LIN {X 0.112,Y -477.429,Z 574.534,A 0.000,B 0.000,C 90.000,E1 96.144} C_DIS
LIN {X 0.154,Y -458.820,Z 574.520,A 0.000,B 0.000,C 90.000,E1 93.612} C_DIS
LIN {X 0.164,Y -448.919,Z 574.512,A 0.000,B 0.000,C 90.000,E1 92.064} C_DIS
LIN {X -0.078,Y -437.148,Z 574.500,A 0.000,B 0.000,C 90.000,E1 90.000} C_DIS
LIN {X -0.153,Y -429.554,Z 574.493,A 0.000,B 0.000,C 90.000,E1 88.682} C_DIS
LIN {X -0.207,Y -419.996,Z 574.484,A 0.000,B 0.000,C 90.000,E1 87.078} C_DIS
LIN {X -0.150,Y -405.811,Z 574.470,A 0.000,B 0.000,C 90.000,E1 84.609} C_DIS
LIN {X 0.053,Y -392.137,Z 574.456,A 0.000,B 0.000,C 90.000,E1 82.064} C_DIS
LIN {X -0.071,Y -380.234,Z 574.443,A 0.000,B 0.000,C 90.000,E1 79.803} C_DIS
LIN {X 0.033,Y -369.905,Z 574.432,A 0.000,B 0.000,C 90.000,E1 77.757} C_DIS
LIN {X -0.039,Y -355.862,Z 574.416,A 0.000,B 0.000,C 90.000,E1 74.810} C_DIS
LIN {X 0.162,Y -345.723,Z 574.402,A 0.000,B 0.000,C 90.000,E1 72.362} C_DIS
LIN {X -0.128,Y -334.343,Z 574.385,A 0.000,B 0.000,C 90.000,E1 69.337} C_DIS
LIN {X 0.102,Y -322.277,Z 574.364,A 0.000,B 0.000,C 90.000,E1 65.537} C_DIS
LIN {X 0.039,Y -314.723,Z 574.350,A 0.000,B 0.000,C 90.000,E1 62.999} C_DIS
LIN {X 0.116,Y -309.189,Z 574.339,A 0.000,B 0.000,C 90.000,E1 61.051} C_DIS
LIN {X 0.043,Y -301.821,Z 574.325,A 0.000,B 0.000,C 90.000,E1 58.456} C_DIS
LIN {X -0.131,Y -293.043,Z 574.306,A 0.000,B 0.000,C 90.000,E1 55.182} C_DIS
LIN {X -0.027,Y -286.344,Z 574.292,A 0.000,B 0.000,C 90.000,E1 52.477} C_DIS
LIN {X -0.003,Y -281.279,Z 574.280,A 0.000,B 0.000,C 90.000,E1 50.436} C_DIS
LIN {X 0.057,Y -277.727,Z 574.273,A 0.000,B 0.000,C 90.000,E1 49.057} C_DIS
LIN {X -0.110,Y -273.909,Z 574.265,A 0.000,B 0.000,C 90.000,E1 47.715} C_DIS
LIN {X 0.043,Y -269.773,Z 574.257,A 0.000,B 0.000,C 90.000,E1 46.296} C_DIS
LIN {X 0.008,Y -264.223,Z 574.248,A 0.000,B 0.000,C 90.000,E1 44.555} C_DIS
LIN {X -0.039,Y -256.042,Z 574.234,A 0.000,B 0.000,C 90.000,E1 42.081} C_DIS
LIN {X -0.053,Y -247.040,Z 574.218,A 0.000,B 0.000,C 90.000,E1 39.197} C_DIS
LIN {X -0.005,Y -238.686,Z 574.201,A 0.000,B 0.000,C 90.000,E1 36.251} C_DIS
LIN {X -0.102,Y -231.066,Z 574.185,A 0.000,B 0.000,C 90.000,E1 33.293} C_DIS
LIN {X -0.069,Y -224.084,Z 574.168,A 0.000,B 0.000,C 90.000,E1 30.256} C_DIS
LIN {X -0.051,Y -217.874,Z 574.151,A 0.000,B 0.000,C 90.000,E1 27.180} C_DIS
LIN {X 0.042,Y -211.020,Z 574.129,A 0.000,B 0.000,C 90.000,E1 23.259} C_DIS
LIN {X -0.047,Y -207.521,Z 574.116,A 0.000,B 0.000,C 90.000,E1 20.918} C_DIS
LIN {X 0.044,Y -203.153,Z 574.094,A 0.000,B 0.000,C 90.000,E1 16.913} C_DIS
LIN {X -0.057,Y -199.050,Z 574.067,A 0.000,B 0.000,C 90.000,E1 12.119} C_DIS
LIN {X -0.009,Y -196.173,Z 574.036,A 0.000,B 0.000,C 90.000,E1 6.429} C_DIS
LIN {X 0.096,Y -197.227,Z 573.966,A 0.000,B 0.000,C 90.000,E1 353.799} C_DIS
LIN {X 0.117,Y -200.242,Z 573.939,A 0.000,B 0.000,C 90.000,E1 348.926} C_DIS
LIN {X -0.103,Y -204.574,Z 573.912,A 0.000,B 0.000,C 90.000,E1 344.157} C_DIS
LIN {X 0.013,Y -209.015,Z 573.890,A 0.000,B 0.000,C 90.000,E1 340.134} C_DIS
LIN {X 0.040,Y -214.221,Z 573.868,A 0.000,B 0.000,C 90.000,E1 336.177} C_DIS
LIN {X 0.003,Y -220.034,Z 573.846,A 0.000,B 0.000,C 90.000,E1 332.281} C_DIS
LIN {X 0.073,Y -226.533,Z 573.825,A 0.000,B 0.000,C 90.000,E1 328.408} C_DIS
LIN {X 0.054,Y -233.497,Z 573.803,A 0.000,B 0.000,C 90.000,E1 324.609} C_DIS
LIN {X -0.045,Y -240.933,Z 573.783,A 0.000,B 0.000,C 90.000,E1 320.884} C_DIS
LIN {X -0.024,Y -249.035,Z 573.762,A 0.000,B 0.000,C 90.000,E1 317.187} C_DIS
LIN {X 0.039,Y -258.163,Z 573.742,A 0.000,B 0.000,C 90.000,E1 313.542} C_DIS
LIN {X 0.041,Y -267.648,Z 573.724,A 0.000,B 0.000,C 90.000,E1 310.334} C_DIS
LIN {X -0.022,Y -278.544,Z 573.707,A 0.000,B 0.000,C 90.000,E1 307.202} C_DIS
LIN {X 0.000,Y -290.576,Z 573.690,A 0.000,B 0.000,C 90.000,E1 304.119} C_DIS
LIN {X -0.128,Y -302.311,Z 573.675,A 0.000,B 0.000,C 90.000,E1 301.465} C_DIS
LIN {X 0.107,Y -317.954,Z 573.656,A 0.000,B 0.000,C 90.000,E1 298.153} C_DIS
LIN {X 0.082,Y -329.625,Z 573.644,A 0.000,B 0.000,C 90.000,E1 295.924} C_DIS
LIN {X 0.018,Y -346.174,Z 573.629,A 0.000,B 0.000,C 90.000,E1 293.131} C_DIS
LIN {X -0.193,Y -362.562,Z 573.615,A 0.000,B 0.000,C 90.000,E1 290.737} C_DIS
LIN {X 0.006,Y -385.100,Z 573.599,A 0.000,B 0.000,C 90.000,E1 287.764} C_DIS
LIN {X 0.185,Y -399.349,Z 573.589,A 0.000,B 0.000,C 90.000,E1 286.024} C_DIS
LIN {X -0.165,Y -416.052,Z 573.578,A 0.000,B 0.000,C 90.000,E1 284.120} C_DIS
LIN {X 0.124,Y -427.790,Z 573.571,A 0.000,B 0.000,C 90.000,E1 282.715} C_DIS
LIN {X -0.014,Y -436.730,Z 573.565,A 0.000,B 0.000,C 90.000,E1 281.658} C_DIS
LIN {X 0.166,Y -447.196,Z 573.557,A 0.000,B 0.000,C 90.000,E1 280.310} C_DIS
LIN {X 0.167,Y -454.942,Z 573.552,A 0.000,B 0.000,C 90.000,E1 279.265} C_DIS
LIN {X -0.198,Y -462.088,Z 573.546,A 0.000,B 0.000,C 90.000,E1 278.276} C_DIS
LIN {X 0.076,Y -467.087,Z 573.542,A 0.000,B 0.000,C 90.000,E1 277.473} C_DIS
LIN {X -0.163,Y -473.101,Z 573.536,A 0.000,B 0.000,C 90.000,E1 276.486} C_DIS
LIN {X 0.221,Y -477.051,Z 573.532,A 0.000,B 0.000,C 90.000,E1 275.682} C_DIS
LIN {X -0.118,Y -479.359,Z 573.529,A 0.000,B 0.000,C 90.000,E1 275.220} C_DIS
LIN {X 0.032,Y -481.383,Z 573.526,A 0.000,B 0.000,C 90.000,E1 274.702} C_DIS
LIN {X 0.152,Y -483.121,Z 573.523,A 0.000,B 0.000,C 90.000,E1 274.188} C_DIS
LIN {X -0.162,Y -484.557,Z 573.521,A 0.000,B 0.000,C 90.000,E1 273.726} C_DIS
LIN {X -0.014,Y -485.710,Z 573.518,A 0.000,B 0.000,C 90.000,E1 273.212} C_DIS
LIN {X 0.169,Y -486.537,Z 573.515,A 0.000,B 0.000,C 90.000,E1 272.694} C_DIS
LIN {X -0.150,Y -487.006,Z 573.512,A 0.000,B 0.000,C 90.000,E1 272.236} C_DIS
LIN {X 0.039,Y -487.014,Z 573.510,A 0.000,B 0.000,C 90.000,E1 271.718} C_DIS
LIN {X 0.214,Y -486.589,Z 573.507,A 0.000,B 0.000,C 90.000,E1 271.203} C_DIS
LIN {X -0.096,Y -485.650,Z 573.504,A 0.000,B 0.000,C 90.000,E1 270.745} C_DIS
LIN {X 0.079,Y -484.122,Z 573.501,A 0.000,B 0.000,C 90.000,E1 270.229} C_DIS
LIN {X -0.235,Y -481.976,Z 573.499,A 0.000,B 0.000,C 90.000,E1 269.771} C_DIS
LIN {X -0.076,Y -479.155,Z 573.496,A 0.000,B 0.000,C 90.000,E1 269.255} C_DIS
LIN {X 0.062,Y -475.438,Z 573.493,A 0.000,B 0.000,C 90.000,E1 268.740} C_DIS
LIN {X -0.116,Y -473.227,Z 573.492,A 0.000,B 0.000,C 90.000,E1 268.511} C_DIS
LIN {X 0.055,Y -467.994,Z 573.489,A 0.000,B 0.000,C 90.000,E1 267.993} C_DIS
LIN {X -0.080,Y -464.987,Z 573.488,A 0.000,B 0.000,C 90.000,E1 267.764} C_DIS
LIN {X 0.012,Y -461.927,Z 573.486,A 0.000,B 0.000,C 90.000,E1 267.535} C_DIS
LIN {X 0.103,Y -458.461,Z 573.485,A 0.000,B 0.000,C 90.000,E1 267.306} C_DIS
LIN {X -0.021,Y -451.459,Z 573.483,A 0.000,B 0.000,C 90.000,E1 266.963} C_DIS
LIN {X -0.030,Y -444.190,Z 573.482,A 0.000,B 0.000,C 90.000,E1 266.674} C_DIS
LIN {X -0.063,Y -436.219,Z 573.480,A 0.000,B 0.000,C 90.000,E1 266.445} C_DIS
LIN {X -0.029,Y -428.400,Z 573.479,A 0.000,B 0.000,C 90.000,E1 266.274} C_DIS
LIN {X -0.099,Y -418.799,Z 573.479,A 0.000,B 0.000,C 90.000,E1 266.159} C_DIS
LIN {X -0.138,Y -408.823,Z 573.478,A 0.000,B 0.000,C 90.000,E1 266.102} C_DIS
LIN {X -0.094,Y -180.923,Z 573.478,A 0.000,B 0.000,C 90.000,E1 266.102} C_DIS
LIN {X -0.052,Y -180.872,Z 573.472,A 0.000,B 0.000,C 90.000,E1 265.065} C_DIS
LIN {X 0.032,Y -178.936,Z 573.443,A 0.000,B 0.000,C 90.000,E1 259.803} C_DIS
LIN {X 0.069,Y -175.984,Z 573.415,A 0.000,B 0.000,C 90.000,E1 254.700} C_DIS
LIN {X 0.014,Y -175.481,Z 573.410,A 0.000,B 0.000,C 90.000,E1 253.866} C_DIS
LIN {X 0.070,Y -172.226,Z 573.387,A 0.000,B 0.000,C 90.000,E1 249.571} C_DIS
LIN {X 0.048,Y -171.703,Z 573.382,A 0.000,B 0.000,C 90.000,E1 248.720} C_DIS
LIN {X -0.027,Y -167.298,Z 573.353,A 0.000,B 0.000,C 90.000,E1 243.563} C_DIS
LIN {X 0.055,Y -166.676,Z 573.348,A 0.000,B 0.000,C 90.000,E1 242.666} C_DIS
LIN {X -0.029,Y -162.658,Z 573.324,A 0.000,B 0.000,C 90.000,E1 238.329} C_DIS
LIN {X 0.033,Y -161.348,Z 573.314,A 0.000,B 0.000,C 90.000,E1 236.548} C_DIS
LIN {X 0.075,Y -157.342,Z 573.290,A 0.000,B 0.000,C 90.000,E1 232.110} C_DIS
LIN {X 0.008,Y -155.328,Z 573.275,A 0.000,B 0.000,C 90.000,E1 229.461} C_DIS
LIN {X -0.062,Y -151.679,Z 573.250,A 0.000,B 0.000,C 90.000,E1 225.000} C_DIS
LIN {X -0.014,Y -150.543,Z 573.240,A 0.000,B 0.000,C 90.000,E1 223.176} C_DIS
LIN {X 0.019,Y -147.269,Z 573.215,A 0.000,B 0.000,C 90.000,E1 218.624} C_DIS
LIN {X -0.008,Y -145.296,Z 573.194,A 0.000,B 0.000,C 90.000,E1 214.978} C_DIS
LIN {X -0.016,Y -142.392,Z 573.164,A 0.000,B 0.000,C 90.000,E1 209.461} C_DIS
LIN {X 0.031,Y -141.372,Z 573.148,A 0.000,B 0.000,C 90.000,E1 206.668} C_DIS
LIN {X 0.008,Y -139.346,Z 573.112,A 0.000,B 0.000,C 90.000,E1 200.174} C_DIS
LIN {X 0.013,Y -139.018,Z 573.102,A 0.000,B 0.000,C 90.000,E1 198.308} C_DIS
LIN {X 0.009,Y -138.343,Z 573.055,A 0.000,B 0.000,C 90.000,E1 189.905} C_DIS
LIN {X 0.029,Y -139.392,Z 573.008,A 0.000,B 0.000,C 90.000,E1 181.489} C_DIS
LIN {X -0.058,Y -141.291,Z 572.972,A 0.000,B 0.000,C 90.000,E1 175.008} C_DIS
LIN {X 0.041,Y -142.654,Z 572.957,A 0.000,B 0.000,C 90.000,E1 172.186} C_DIS
LIN {X -0.009,Y -144.994,Z 572.931,A 0.000,B 0.000,C 90.000,E1 167.589} C_DIS
LIN {X -0.020,Y -147.621,Z 572.911,A 0.000,B 0.000,C 90.000,E1 163.921} C_DIS
LIN {X 0.059,Y -150.248,Z 572.890,A 0.000,B 0.000,C 90.000,E1 160.242} C_DIS
LIN {X -0.068,Y -153.643,Z 572.870,A 0.000,B 0.000,C 90.000,E1 156.666} C_DIS
LIN {X -0.010,Y -157.059,Z 572.850,A 0.000,B 0.000,C 90.000,E1 153.050} C_DIS
LIN {X 0.070,Y -161.189,Z 572.830,A 0.000,B 0.000,C 90.000,E1 149.459} C_DIS
LIN {X 0.018,Y -163.282,Z 572.821,A 0.000,B 0.000,C 90.000,E1 147.709} C_DIS
LIN {X 0.029,Y -167.726,Z 572.801,A 0.000,B 0.000,C 90.000,E1 144.196} C_DIS
LIN {X -0.059,Y -171.544,Z 572.787,A 0.000,B 0.000,C 90.000,E1 141.618} C_DIS
LIN {X -0.017,Y -176.487,Z 572.768,A 0.000,B 0.000,C 90.000,E1 138.162} C_DIS
LIN {X 0.109,Y -180.784,Z 572.753,A 0.000,B 0.000,C 90.000,E1 135.567} C_DIS
LIN {X -0.030,Y -186.190,Z 572.735,A 0.000,B 0.000,C 90.000,E1 132.243} C_DIS
LIN {X -0.047,Y -191.398,Z 572.719,A 0.000,B 0.000,C 90.000,E1 129.402} C_DIS
LIN {X 0.021,Y -191.570,Z 572.718,A 0.000,B 0.000,C 90.000,E1 129.277} C_DIS
LIN {X -0.003,Y -288.514,Z 572.718,A 0.000,B 0.000,C 90.000,E1 129.277} C_DIS
LIN {X -0.139,Y -294.073,Z 572.717,A 0.000,B 0.000,C 90.000,E1 129.116} C_DIS
LIN {X -0.012,Y -296.456,Z 572.716,A 0.000,B 0.000,C 90.000,E1 128.910} C_DIS
LIN {X -0.037,Y -300.301,Z 572.714,A 0.000,B 0.000,C 90.000,E1 128.463} C_DIS
LIN {X -0.032,Y -302.189,Z 572.712,A 0.000,B 0.000,C 90.000,E1 128.141} C_DIS
LIN {X 0.024,Y -303.668,Z 572.710,A 0.000,B 0.000,C 90.000,E1 127.810} C_DIS
LIN {X -0.019,Y -304.870,Z 572.708,A 0.000,B 0.000,C 90.000,E1 127.488} C_DIS
LIN {X -0.102,Y -315.567,Z 572.688,A 0.000,B 0.000,C 90.000,E1 123.913} C_DIS
LIN {X 0.048,Y -325.634,Z 572.672,A 0.000,B 0.000,C 90.000,E1 121.003} C_DIS
LIN {X -0.002,Y -337.035,Z 572.657,A 0.000,B 0.000,C 90.000,E1 118.180} C_DIS
LIN {X -0.037,Y -349.867,Z 572.641,A 0.000,B 0.000,C 90.000,E1 115.412} C_DIS
LIN {X -0.085,Y -362.572,Z 572.628,A 0.000,B 0.000,C 90.000,E1 113.003} C_DIS
LIN {X 0.097,Y -376.592,Z 572.615,A 0.000,B 0.000,C 90.000,E1 110.610} C_DIS
LIN {X 0.033,Y -392.029,Z 572.602,A 0.000,B 0.000,C 90.000,E1 108.308} C_DIS
LIN {X -0.155,Y -408.997,Z 572.589,A 0.000,B 0.000,C 90.000,E1 106.079} C_DIS
LIN {X -0.169,Y -427.620,Z 572.577,A 0.000,B 0.000,C 90.000,E1 103.883} C_DIS
LIN {X 0.000,Y -447.571,Z 572.565,A 0.000,B 0.000,C 90.000,E1 101.771} C_DIS
LIN {X 0.033,Y -468.110,Z 572.555,A 0.000,B 0.000,C 90.000,E1 99.849} C_DIS
LIN {X 0.173,Y -473.326,Z 572.552,A 0.000,B 0.000,C 90.000,E1 99.378} C_DIS
LIN {X 0.186,Y -475.660,Z 572.551,A 0.000,B 0.000,C 90.000,E1 99.151} C_DIS
LIN {X 0.141,Y -477.532,Z 572.550,A 0.000,B 0.000,C 90.000,E1 98.916} C_DIS
LIN {X 0.095,Y -478.953,Z 572.548,A 0.000,B 0.000,C 90.000,E1 98.681} C_DIS
LIN {X 0.241,Y -480.865,Z 572.546,A 0.000,B 0.000,C 90.000,E1 98.163} C_DIS
LIN {X -0.081,Y -481.662,Z 572.543,A 0.000,B 0.000,C 90.000,E1 97.701} C_DIS
LIN {X 0.086,Y -481.478,Z 572.540,A 0.000,B 0.000,C 90.000,E1 97.182} C_DIS
LIN {X -0.219,Y -480.290,Z 572.537,A 0.000,B 0.000,C 90.000,E1 96.720} C_DIS
LIN {X 0.132,Y -479.262,Z 572.536,A 0.000,B 0.000,C 90.000,E1 96.429} C_DIS
LIN {X -0.047,Y -477.879,Z 572.534,A 0.000,B 0.000,C 90.000,E1 96.201} C_DIS
LIN {X -0.055,Y -462.852,Z 572.523,A 0.000,B 0.000,C 90.000,E1 94.188} C_DIS
LIN {X 0.053,Y -452.448,Z 572.515,A 0.000,B 0.000,C 90.000,E1 92.636} C_DIS
LIN {X 0.142,Y -441.852,Z 572.505,A 0.000,B 0.000,C 90.000,E1 90.802} C_DIS
LIN {X 0.136,Y -434.485,Z 572.497,A 0.000,B 0.000,C 90.000,E1 89.484} C_DIS
LIN {X 0.030,Y -426.727,Z 572.490,A 0.000,B 0.000,C 90.000,E1 88.165} C_DIS
LIN {X 0.123,Y -413.943,Z 572.478,A 0.000,B 0.000,C 90.000,E1 85.988} C_DIS
LIN {X 0.001,Y -401.487,Z 572.466,A 0.000,B 0.000,C 90.000,E1 83.799} C_DIS
LIN {X 0.040,Y -389.431,Z 572.453,A 0.000,B 0.000,C 90.000,E1 81.546} C_DIS
LIN {X -0.083,Y -377.555,Z 572.440,A 0.000,B 0.000,C 90.000,E1 79.275} C_DIS
LIN {X -0.063,Y -364.322,Z 572.426,A 0.000,B 0.000,C 90.000,E1 76.645} C_DIS
LIN {X -0.092,Y -353.407,Z 572.413,A 0.000,B 0.000,C 90.000,E1 74.267} C_DIS
LIN {X 0.056,Y -343.521,Z 572.399,A 0.000,B 0.000,C 90.000,E1 71.819} C_DIS
LIN {X 0.132,Y -332.421,Z 572.382,A 0.000,B 0.000,C 90.000,E1 68.720} C_DIS
LIN {X -0.003,Y -320.547,Z 572.361,A 0.000,B 0.000,C 90.000,E1 64.973} C_DIS
LIN {X 0.033,Y -313.070,Z 572.347,A 0.000,B 0.000,C 90.000,E1 62.410} C_DIS
LIN {X 0.173,Y -305.663,Z 572.332,A 0.000,B 0.000,C 90.000,E1 59.793} C_DIS
LIN {X -0.046,Y -296.647,Z 572.314,A 0.000,B 0.000,C 90.000,E1 56.548} C_DIS
LIN {X 0.046,Y -289.830,Z 572.299,A 0.000,B 0.000,C 90.000,E1 53.863} C_DIS
LIN {X 0.131,Y -284.820,Z 572.288,A 0.000,B 0.000,C 90.000,E1 51.823} C_DIS
LIN {X -0.091,Y -279.648,Z 572.277,A 0.000,B 0.000,C 90.000,E1 49.828} C_DIS
LIN {X -0.050,Y -275.951,Z 572.269,A 0.000,B 0.000,C 90.000,E1 48.447} C_DIS
LIN {X -0.053,Y -272.012,Z 572.261,A 0.000,B 0.000,C 90.000,E1 47.067} C_DIS
LIN {X -0.043,Y -266.626,Z 572.252,A 0.000,B 0.000,C 90.000,E1 45.324} C_DIS
LIN {X -0.087,Y -259.680,Z 572.240,A 0.000,B 0.000,C 90.000,E1 43.218} C_DIS
LIN {X 0.009,Y -249.341,Z 572.222,A 0.000,B 0.000,C 90.000,E1 39.967} C_DIS
LIN {X 0.066,Y -240.775,Z 572.206,A 0.000,B 0.000,C 90.000,E1 37.030} C_DIS
LIN {X 0.136,Y -231.132,Z 572.185,A 0.000,B 0.000,C 90.000,E1 33.293} C_DIS
LIN {X -0.144,Y -224.123,Z 572.168,A 0.000,B 0.000,C 90.000,E1 30.335} C_DIS
LIN {X -0.118,Y -217.897,Z 572.151,A 0.000,B 0.000,C 90.000,E1 27.257} C_DIS
LIN {X -0.015,Y -211.021,Z 572.130,A 0.000,B 0.000,C 90.000,E1 23.334} C_DIS
LIN {X -0.025,Y -207.515,Z 572.116,A 0.000,B 0.000,C 90.000,E1 20.972} C_DIS
LIN {X 0.003,Y -203.164,Z 572.094,A 0.000,B 0.000,C 90.000,E1 16.985} C_DIS
LIN {X 0.061,Y -199.622,Z 572.072,A 0.000,B 0.000,C 90.000,E1 12.952} C_DIS
LIN {X 0.013,Y -196.446,Z 572.041,A 0.000,B 0.000,C 90.000,E1 7.296} C_DIS
LIN {X 0.095,Y -197.213,Z 571.966,A 0.000,B 0.000,C 90.000,E1 353.799} C_DIS
LIN {X -0.078,Y -200.873,Z 571.934,A 0.000,B 0.000,C 90.000,E1 348.173} C_DIS
LIN {X 0.014,Y -205.397,Z 571.907,A 0.000,B 0.000,C 90.000,E1 343.323} C_DIS
LIN {X 0.027,Y -210.010,Z 571.885,A 0.000,B 0.000,C 90.000,E1 339.337} C_DIS
LIN {X -0.024,Y -215.316,Z 571.863,A 0.000,B 0.000,C 90.000,E1 335.409} C_DIS
LIN {X -0.025,Y -221.258,Z 571.842,A 0.000,B 0.000,C 90.000,E1 331.513} C_DIS
LIN {X 0.070,Y -226.519,Z 571.825,A 0.000,B 0.000,C 90.000,E1 328.408} C_DIS
LIN {X 0.050,Y -233.464,Z 571.803,A 0.000,B 0.000,C 90.000,E1 324.609} C_DIS
LIN {X -0.049,Y -240.913,Z 571.783,A 0.000,B 0.000,C 90.000,E1 320.884} C_DIS
LIN {X 0.139,Y -248.985,Z 571.762,A 0.000,B 0.000,C 90.000,E1 317.148} C_DIS
LIN {X 0.033,Y -258.158,Z 571.742,A 0.000,B 0.000,C 90.000,E1 313.542} C_DIS
LIN {X 0.035,Y -267.655,Z 571.724,A 0.000,B 0.000,C 90.000,E1 310.334} C_DIS
LIN {X -0.029,Y -278.520,Z 571.707,A 0.000,B 0.000,C 90.000,E1 307.202} C_DIS
LIN {X -0.032,Y -291.977,Z 571.688,A 0.000,B 0.000,C 90.000,E1 303.785} C_DIS
LIN {X -0.100,Y -305.268,Z 571.671,A 0.000,B 0.000,C 90.000,E1 300.797} C_DIS
LIN {X 0.081,Y -321.139,Z 571.653,A 0.000,B 0.000,C 90.000,E1 297.513} C_DIS
LIN {X 0.169,Y -331.291,Z 571.642,A 0.000,B 0.000,C 90.000,E1 295.591} C_DIS
LIN {X -0.001,Y -346.091,Z 571.628,A 0.000,B 0.000,C 90.000,E1 293.131} C_DIS
LIN {X 0.195,Y -360.396,Z 571.617,A 0.000,B 0.000,C 90.000,E1 290.972} C_DIS
LIN {X -0.026,Y -382.783,Z 571.600,A 0.000,B 0.000,C 90.000,E1 288.055} C_DIS
LIN {X 0.160,Y -399.346,Z 571.589,A 0.000,B 0.000,C 90.000,E1 286.024} C_DIS
LIN {X -0.190,Y -416.096,Z 571.578,A 0.000,B 0.000,C 90.000,E1 284.120} C_DIS
LIN {X 0.098,Y -427.846,Z 571.571,A 0.000,B 0.000,C 90.000,E1 282.715} C_DIS
LIN {X -0.040,Y -436.797,Z 571.565,A 0.000,B 0.000,C 90.000,E1 281.658} C_DIS
LIN {X 0.140,Y -447.285,Z 571.557,A 0.000,B 0.000,C 90.000,E1 280.310} C_DIS
LIN {X 0.142,Y -455.058,Z 571.552,A 0.000,B 0.000,C 90.000,E1 279.265} C_DIS
LIN {X 0.235,Y -462.192,Z 571.546,A 0.000,B 0.000,C 90.000,E1 278.219} C_DIS
LIN {X 0.053,Y -467.183,Z 571.542,A 0.000,B 0.000,C 90.000,E1 277.473} C_DIS
LIN {X -0.185,Y -473.192,Z 571.536,A 0.000,B 0.000,C 90.000,E1 276.486} C_DIS
LIN {X 0.199,Y -477.113,Z 571.532,A 0.000,B 0.000,C 90.000,E1 275.682} C_DIS
LIN {X -0.139,Y -479.404,Z 571.529,A 0.000,B 0.000,C 90.000,E1 275.220} C_DIS
LIN {X 0.011,Y -481.437,Z 571.526,A 0.000,B 0.000,C 90.000,E1 274.702} C_DIS
LIN {X 0.131,Y -483.178,Z 571.523,A 0.000,B 0.000,C 90.000,E1 274.188} C_DIS
LIN {X -0.183,Y -484.616,Z 571.521,A 0.000,B 0.000,C 90.000,E1 273.726} C_DIS
LIN {X -0.035,Y -485.757,Z 571.518,A 0.000,B 0.000,C 90.000,E1 273.212} C_DIS
LIN {X 0.149,Y -486.563,Z 571.515,A 0.000,B 0.000,C 90.000,E1 272.694} C_DIS
LIN {X -0.171,Y -487.031,Z 571.512,A 0.000,B 0.000,C 90.000,E1 272.236} C_DIS
LIN {X 0.019,Y -487.045,Z 571.510,A 0.000,B 0.000,C 90.000,E1 271.718} C_DIS
LIN {X 0.194,Y -486.598,Z 571.507,A 0.000,B 0.000,C 90.000,E1 271.203} C_DIS
LIN {X -0.115,Y -485.613,Z 571.504,A 0.000,B 0.000,C 90.000,E1 270.745} C_DIS
LIN {X 0.059,Y -484.100,Z 571.501,A 0.000,B 0.000,C 90.000,E1 270.229} C_DIS
LIN {X 0.227,Y -481.963,Z 571.499,A 0.000,B 0.000,C 90.000,E1 269.714} C_DIS
LIN {X -0.095,Y -479.106,Z 571.496,A 0.000,B 0.000,C 90.000,E1 269.255} C_DIS
LIN {X 0.042,Y -475.374,Z 571.493,A 0.000,B 0.000,C 90.000,E1 268.740} C_DIS
LIN {X -0.137,Y -473.178,Z 571.492,A 0.000,B 0.000,C 90.000,E1 268.511} C_DIS
LIN {X 0.158,Y -470.693,Z 571.490,A 0.000,B 0.000,C 90.000,E1 268.224} C_DIS
LIN {X -0.140,Y -464.814,Z 571.487,A 0.000,B 0.000,C 90.000,E1 267.764} C_DIS
LIN {X -0.024,Y -461.813,Z 571.486,A 0.000,B 0.000,C 90.000,E1 267.535} C_DIS
LIN {X 0.026,Y -455.147,Z 571.484,A 0.000,B 0.000,C 90.000,E1 267.135} C_DIS
LIN {X 0.213,Y -447.942,Z 571.482,A 0.000,B 0.000,C 90.000,E1 266.788} C_DIS
LIN {X -0.028,Y -440.612,Z 571.481,A 0.000,B 0.000,C 90.000,E1 266.560} C_DIS
LIN {X 0.181,Y -432.743,Z 571.480,A 0.000,B 0.000,C 90.000,E1 266.331} C_DIS
LIN {X -0.044,Y -424.386,Z 571.479,A 0.000,B 0.000,C 90.000,E1 266.216} C_DIS
LIN {X 0.037,Y -414.363,Z 571.478,A 0.000,B 0.000,C 90.000,E1 266.102} C_DIS
LIN {X -0.193,Y -406.159,Z 571.478,A 0.000,B 0.000,C 90.000,E1 266.102} C_DIS
LIN {X 0.060,Y -180.923,Z 571.478,A 0.000,B 0.000,C 90.000,E1 266.045} C_DIS
LIN {X -0.077,Y -180.870,Z 571.472,A 0.000,B 0.000,C 90.000,E1 265.065} C_DIS
LIN {X 0.007,Y -178.932,Z 571.443,A 0.000,B 0.000,C 90.000,E1 259.803} C_DIS
LIN {X 0.044,Y -175.981,Z 571.415,A 0.000,B 0.000,C 90.000,E1 254.700} C_DIS
LIN {X -0.010,Y -175.473,Z 571.410,A 0.000,B 0.000,C 90.000,E1 253.866} C_DIS
LIN {X 0.046,Y -172.221,Z 571.387,A 0.000,B 0.000,C 90.000,E1 249.571} C_DIS
LIN {X 0.023,Y -171.697,Z 571.382,A 0.000,B 0.000,C 90.000,E1 248.720} C_DIS
LIN {X -0.051,Y -167.292,Z 571.353,A 0.000,B 0.000,C 90.000,E1 243.563} C_DIS
LIN {X 0.031,Y -166.669,Z 571.348,A 0.000,B 0.000,C 90.000,E1 242.666} C_DIS
LIN {X -0.053,Y -162.652,Z 571.324,A 0.000,B 0.000,C 90.000,E1 238.329} C_DIS
LIN {X 0.010,Y -161.340,Z 571.314,A 0.000,B 0.000,C 90.000,E1 236.548} C_DIS
LIN {X 0.052,Y -157.335,Z 571.290,A 0.000,B 0.000,C 90.000,E1 232.110} C_DIS
LIN {X -0.015,Y -155.319,Z 571.275,A 0.000,B 0.000,C 90.000,E1 229.461} C_DIS
LIN {X 0.022,Y -151.673,Z 571.250,A 0.000,B 0.000,C 90.000,E1 224.960} C_DIS
LIN {X -0.036,Y -150.538,Z 571.240,A 0.000,B 0.000,C 90.000,E1 223.176} C_DIS
LIN {X -0.004,Y -147.263,Z 571.215,A 0.000,B 0.000,C 90.000,E1 218.624} C_DIS
LIN {X -0.030,Y -145.290,Z 571.194,A 0.000,B 0.000,C 90.000,E1 214.978} C_DIS
LIN {X -0.037,Y -142.388,Z 571.164,A 0.000,B 0.000,C 90.000,E1 209.461} C_DIS
LIN {X 0.008,Y -141.368,Z 571.148,A 0.000,B 0.000,C 90.000,E1 206.668} C_DIS
LIN {X -0.013,Y -139.344,Z 571.112,A 0.000,B 0.000,C 90.000,E1 200.174} C_DIS
LIN {X -0.008,Y -139.015,Z 571.102,A 0.000,B 0.000,C 90.000,E1 198.308} C_DIS
LIN {X -0.012,Y -138.342,Z 571.055,A 0.000,B 0.000,C 90.000,E1 189.905} C_DIS
LIN {X 0.007,Y -139.394,Z 571.008,A 0.000,B 0.000,C 90.000,E1 181.489} C_DIS
LIN {X 0.061,Y -141.296,Z 570.972,A 0.000,B 0.000,C 90.000,E1 174.951} C_DIS
LIN {X 0.019,Y -142.657,Z 570.957,A 0.000,B 0.000,C 90.000,E1 172.186} C_DIS
LIN {X -0.031,Y -145.000,Z 570.931,A 0.000,B 0.000,C 90.000,E1 167.589} C_DIS
LIN {X -0.042,Y -147.627,Z 570.911,A 0.000,B 0.000,C 90.000,E1 163.921} C_DIS
LIN {X 0.036,Y -150.255,Z 570.890,A 0.000,B 0.000,C 90.000,E1 160.242} C_DIS
LIN {X 0.050,Y -153.653,Z 570.870,A 0.000,B 0.000,C 90.000,E1 156.613} C_DIS
LIN {X -0.033,Y -157.067,Z 570.850,A 0.000,B 0.000,C 90.000,E1 153.050} C_DIS
LIN {X 0.046,Y -161.200,Z 570.830,A 0.000,B 0.000,C 90.000,E1 149.459} C_DIS
LIN {X -0.005,Y -163.292,Z 570.821,A 0.000,B 0.000,C 90.000,E1 147.709} C_DIS
LIN {X 0.005,Y -167.737,Z 570.801,A 0.000,B 0.000,C 90.000,E1 144.196} C_DIS
LIN {X -0.083,Y -171.555,Z 570.787,A 0.000,B 0.000,C 90.000,E1 141.618} C_DIS
LIN {X -0.042,Y -176.499,Z 570.768,A 0.000,B 0.000,C 90.000,E1 138.162} C_DIS
LIN {X 0.083,Y -180.796,Z 570.753,A 0.000,B 0.000,C 90.000,E1 135.567} C_DIS
LIN {X 0.069,Y -186.204,Z 570.735,A 0.000,B 0.000,C 90.000,E1 132.204} C_DIS
LIN {X 0.075,Y -191.412,Z 570.719,A 0.000,B 0.000,C 90.000,E1 129.358} C_DIS
LIN {X -0.029,Y -191.594,Z 570.718,A 0.000,B 0.000,C 90.000,E1 129.277} C_DIS
LIN {X -0.079,Y -288.721,Z 570.718,A 0.000,B 0.000,C 90.000,E1 129.277} C_DIS
LIN {X 0.048,Y -294.000,Z 570.717,A 0.000,B 0.000,C 90.000,E1 129.072} C_DIS
LIN {X -0.053,Y -296.411,Z 570.716,A 0.000,B 0.000,C 90.000,E1 128.910} C_DIS
LIN {X -0.054,Y -300.249,Z 570.714,A 0.000,B 0.000,C 90.000,E1 128.463} C_DIS
LIN {X -0.038,Y -302.142,Z 570.712,A 0.000,B 0.000,C 90.000,E1 128.141} C_DIS
LIN {X 0.029,Y -303.627,Z 570.710,A 0.000,B 0.000,C 90.000,E1 127.810} C_DIS
LIN {X -0.015,Y -304.840,Z 570.708,A 0.000,B 0.000,C 90.000,E1 127.488} C_DIS
LIN {X -0.098,Y -315.543,Z 570.688,A 0.000,B 0.000,C 90.000,E1 123.913} C_DIS
LIN {X 0.052,Y -325.610,Z 570.672,A 0.000,B 0.000,C 90.000,E1 121.003} C_DIS
LIN {X 0.001,Y -337.011,Z 570.657,A 0.000,B 0.000,C 90.000,E1 118.180} C_DIS
LIN {X -0.035,Y -349.843,Z 570.641,A 0.000,B 0.000,C 90.000,E1 115.412} C_DIS
LIN {X -0.084,Y -362.547,Z 570.628,A 0.000,B 0.000,C 90.000,E1 113.003} C_DIS
LIN {X 0.098,Y -376.567,Z 570.615,A 0.000,B 0.000,C 90.000,E1 110.610} C_DIS
LIN {X 0.033,Y -392.004,Z 570.602,A 0.000,B 0.000,C 90.000,E1 108.308} C_DIS
LIN {X -0.156,Y -408.971,Z 570.589,A 0.000,B 0.000,C 90.000,E1 106.079} C_DIS
LIN {X -0.171,Y -427.593,Z 570.577,A 0.000,B 0.000,C 90.000,E1 103.883} C_DIS
LIN {X -0.002,Y -447.545,Z 570.565,A 0.000,B 0.000,C 90.000,E1 101.771} C_DIS
LIN {X 0.031,Y -468.084,Z 570.555,A 0.000,B 0.000,C 90.000,E1 99.849} C_DIS
LIN {X 0.170,Y -473.299,Z 570.552,A 0.000,B 0.000,C 90.000,E1 99.378} C_DIS
LIN {X 0.183,Y -475.668,Z 570.551,A 0.000,B 0.000,C 90.000,E1 99.151} C_DIS
LIN {X 0.156,Y -477.554,Z 570.550,A 0.000,B 0.000,C 90.000,E1 98.916} C_DIS
LIN {X 0.128,Y -478.989,Z 570.548,A 0.000,B 0.000,C 90.000,E1 98.681} C_DIS
LIN {X -0.203,Y -480.946,Z 570.546,A 0.000,B 0.000,C 90.000,E1 98.219} C_DIS
LIN {X -0.049,Y -481.779,Z 570.543,A 0.000,B 0.000,C 90.000,E1 97.701} C_DIS
LIN {X 0.120,Y -481.632,Z 570.540,A 0.000,B 0.000,C 90.000,E1 97.182} C_DIS
LIN {X -0.185,Y -480.481,Z 570.537,A 0.000,B 0.000,C 90.000,E1 96.720} C_DIS
LIN {X 0.167,Y -479.477,Z 570.536,A 0.000,B 0.000,C 90.000,E1 96.429} C_DIS
LIN {X -0.012,Y -478.121,Z 570.534,A 0.000,B 0.000,C 90.000,E1 96.201} C_DIS
LIN {X -0.186,Y -470.566,Z 570.529,A 0.000,B 0.000,C 90.000,E1 95.220} C_DIS
LIN {X -0.167,Y -457.706,Z 570.519,A 0.000,B 0.000,C 90.000,E1 93.440} C_DIS
LIN {X 0.075,Y -449.432,Z 570.512,A 0.000,B 0.000,C 90.000,E1 92.121} C_DIS
LIN {X 0.014,Y -436.098,Z 570.499,A 0.000,B 0.000,C 90.000,E1 89.771} C_DIS
LIN {X -0.075,Y -428.417,Z 570.491,A 0.000,B 0.000,C 90.000,E1 88.453} C_DIS
LIN {X -0.024,Y -417.227,Z 570.481,A 0.000,B 0.000,C 90.000,E1 86.560} C_DIS
LIN {X -0.097,Y -404.672,Z 570.469,A 0.000,B 0.000,C 90.000,E1 84.375} C_DIS
LIN {X -0.032,Y -392.529,Z 570.456,A 0.000,B 0.000,C 90.000,E1 82.129} C_DIS
LIN {X -0.089,Y -380.575,Z 570.444,A 0.000,B 0.000,C 90.000,E1 79.859} C_DIS
LIN {X 0.025,Y -370.169,Z 570.432,A 0.000,B 0.000,C 90.000,E1 77.813} C_DIS
LIN {X -0.037,Y -356.004,Z 570.416,A 0.000,B 0.000,C 90.000,E1 74.866} C_DIS
LIN {X 0.101,Y -343.525,Z 570.399,A 0.000,B 0.000,C 90.000,E1 71.819} C_DIS
LIN {X -0.132,Y -332.452,Z 570.382,A 0.000,B 0.000,C 90.000,E1 68.773} C_DIS
LIN {X 0.042,Y -320.597,Z 570.361,A 0.000,B 0.000,C 90.000,E1 64.973} C_DIS
LIN {X 0.077,Y -313.103,Z 570.347,A 0.000,B 0.000,C 90.000,E1 62.410} C_DIS
LIN {X 0.063,Y -305.707,Z 570.332,A 0.000,B 0.000,C 90.000,E1 59.822} C_DIS
LIN {X -0.001,Y -296.690,Z 570.314,A 0.000,B 0.000,C 90.000,E1 56.548} C_DIS
LIN {X -0.144,Y -289.845,Z 570.299,A 0.000,B 0.000,C 90.000,E1 53.909} C_DIS
LIN {X 0.176,Y -284.836,Z 570.288,A 0.000,B 0.000,C 90.000,E1 51.823} C_DIS
LIN {X -0.048,Y -279.652,Z 570.277,A 0.000,B 0.000,C 90.000,E1 49.828} C_DIS
LIN {X -0.006,Y -275.942,Z 570.269,A 0.000,B 0.000,C 90.000,E1 48.447} C_DIS
LIN {X -0.010,Y -272.002,Z 570.261,A 0.000,B 0.000,C 90.000,E1 47.067} C_DIS
LIN {X -0.002,Y -266.581,Z 570.252,A 0.000,B 0.000,C 90.000,E1 45.324} C_DIS
LIN {X 0.095,Y -260.809,Z 570.242,A 0.000,B 0.000,C 90.000,E1 43.542} C_DIS
LIN {X 0.023,Y -250.411,Z 570.224,A 0.000,B 0.000,C 90.000,E1 40.334} C_DIS
LIN {X -0.091,Y -240.723,Z 570.206,A 0.000,B 0.000,C 90.000,E1 37.076} C_DIS
LIN {X 0.051,Y -232.930,Z 570.189,A 0.000,B 0.000,C 90.000,E1 34.072} C_DIS
LIN {X 0.059,Y -225.742,Z 570.173,A 0.000,B 0.000,C 90.000,E1 31.052} C_DIS
LIN {X -0.078,Y -219.309,Z 570.156,A 0.000,B 0.000,C 90.000,E1 28.025} C_DIS
LIN {X -0.041,Y -212.269,Z 570.134,A 0.000,B 0.000,C 90.000,E1 24.131} C_DIS
LIN {X -0.029,Y -208.526,Z 570.121,A 0.000,B 0.000,C 90.000,E1 21.770} C_DIS
LIN {X -0.102,Y -203.938,Z 570.099,A 0.000,B 0.000,C 90.000,E1 17.819} C_DIS
LIN {X -0.114,Y -199.568,Z 570.072,A 0.000,B 0.000,C 90.000,E1 13.008} C_DIS
LIN {X 0.029,Y -196.416,Z 570.041,A 0.000,B 0.000,C 90.000,E1 7.296} C_DIS
LIN {X 0.094,Y -197.196,Z 569.966,A 0.000,B 0.000,C 90.000,E1 353.799} C_DIS
LIN {X -0.079,Y -200.859,Z 569.934,A 0.000,B 0.000,C 90.000,E1 348.173} C_DIS
LIN {X 0.012,Y -205.384,Z 569.907,A 0.000,B 0.000,C 90.000,E1 343.323} C_DIS
LIN {X 0.025,Y -210.016,Z 569.885,A 0.000,B 0.000,C 90.000,E1 339.337} C_DIS
LIN {X -0.027,Y -215.307,Z 569.863,A 0.000,B 0.000,C 90.000,E1 335.409} C_DIS
LIN {X -0.028,Y -221.248,Z 569.842,A 0.000,B 0.000,C 90.000,E1 331.513} C_DIS
LIN {X 0.066,Y -226.500,Z 569.825,A 0.000,B 0.000,C 90.000,E1 328.408} C_DIS
LIN {X 0.046,Y -233.434,Z 569.803,A 0.000,B 0.000,C 90.000,E1 324.609} C_DIS
LIN {X -0.055,Y -240.894,Z 569.783,A 0.000,B 0.000,C 90.000,E1 320.884} C_DIS
LIN {X 0.133,Y -248.937,Z 569.762,A 0.000,B 0.000,C 90.000,E1 317.148} C_DIS
LIN {X 0.025,Y -258.149,Z 569.742,A 0.000,B 0.000,C 90.000,E1 313.542} C_DIS
LIN {X 0.032,Y -267.663,Z 569.724,A 0.000,B 0.000,C 90.000,E1 310.334} C_DIS
LIN {X -0.031,Y -278.489,Z 569.707,A 0.000,B 0.000,C 90.000,E1 307.202} C_DIS
LIN {X -0.035,Y -291.930,Z 569.688,A 0.000,B 0.000,C 90.000,E1 303.785} C_DIS
LIN {X -0.106,Y -305.195,Z 569.671,A 0.000,B 0.000,C 90.000,E1 300.797} C_DIS
LIN {X 0.073,Y -321.042,Z 569.653,A 0.000,B 0.000,C 90.000,E1 297.513} C_DIS
LIN {X 0.118,Y -332.976,Z 569.641,A 0.000,B 0.000,C 90.000,E1 295.283} C_DIS
LIN {X -0.014,Y -345.992,Z 569.628,A 0.000,B 0.000,C 90.000,E1 293.131} C_DIS
LIN {X 0.179,Y -360.351,Z 569.617,A 0.000,B 0.000,C 90.000,E1 290.972} C_DIS
LIN {X -0.044,Y -382.768,Z 569.600,A 0.000,B 0.000,C 90.000,E1 288.055} C_DIS
LIN {X 0.142,Y -399.333,Z 569.589,A 0.000,B 0.000,C 90.000,E1 286.024} C_DIS
LIN {X 0.193,Y -416.133,Z 569.578,A 0.000,B 0.000,C 90.000,E1 284.064} C_DIS
LIN {X 0.079,Y -427.893,Z 569.571,A 0.000,B 0.000,C 90.000,E1 282.715} C_DIS
LIN {X -0.059,Y -436.850,Z 569.565,A 0.000,B 0.000,C 90.000,E1 281.658} C_DIS
LIN {X -0.099,Y -445.318,Z 569.559,A 0.000,B 0.000,C 90.000,E1 280.602} C_DIS
LIN {X -0.125,Y -453.242,Z 569.553,A 0.000,B 0.000,C 90.000,E1 279.557} C_DIS
LIN {X -0.056,Y -460.560,Z 569.547,A 0.000,B 0.000,C 90.000,E1 278.511} C_DIS
LIN {X 0.037,Y -467.259,Z 569.542,A 0.000,B 0.000,C 90.000,E1 277.473} C_DIS
LIN {X -0.201,Y -473.259,Z 569.536,A 0.000,B 0.000,C 90.000,E1 276.486} C_DIS
LIN {X 0.183,Y -477.168,Z 569.532,A 0.000,B 0.000,C 90.000,E1 275.682} C_DIS
LIN {X -0.154,Y -479.464,Z 569.529,A 0.000,B 0.000,C 90.000,E1 275.220} C_DIS
LIN {X -0.004,Y -481.470,Z 569.526,A 0.000,B 0.000,C 90.000,E1 274.702} C_DIS
LIN {X 0.117,Y -483.203,Z 569.523,A 0.000,B 0.000,C 90.000,E1 274.188} C_DIS
LIN {X -0.198,Y -484.660,Z 569.521,A 0.000,B 0.000,C 90.000,E1 273.726} C_DIS
LIN {X -0.050,Y -485.799,Z 569.518,A 0.000,B 0.000,C 90.000,E1 273.212} C_DIS
LIN {X 0.135,Y -486.612,Z 569.515,A 0.000,B 0.000,C 90.000,E1 272.694} C_DIS
LIN {X -0.184,Y -487.057,Z 569.512,A 0.000,B 0.000,C 90.000,E1 272.236} C_DIS
LIN {X 0.005,Y -487.059,Z 569.510,A 0.000,B 0.000,C 90.000,E1 271.718} C_DIS
LIN {X 0.181,Y -486.597,Z 569.507,A 0.000,B 0.000,C 90.000,E1 271.203} C_DIS
LIN {X -0.129,Y -485.611,Z 569.504,A 0.000,B 0.000,C 90.000,E1 270.745} C_DIS
LIN {X 0.046,Y -484.056,Z 569.501,A 0.000,B 0.000,C 90.000,E1 270.229} C_DIS
LIN {X 0.214,Y -481.946,Z 569.499,A 0.000,B 0.000,C 90.000,E1 269.714} C_DIS
LIN {X -0.108,Y -479.033,Z 569.496,A 0.000,B 0.000,C 90.000,E1 269.255} C_DIS
LIN {X 0.028,Y -475.349,Z 569.493,A 0.000,B 0.000,C 90.000,E1 268.740} C_DIS
LIN {X -0.150,Y -473.137,Z 569.492,A 0.000,B 0.000,C 90.000,E1 268.511} C_DIS
LIN {X 0.023,Y -467.907,Z 569.489,A 0.000,B 0.000,C 90.000,E1 267.993} C_DIS
LIN {X -0.110,Y -464.853,Z 569.487,A 0.000,B 0.000,C 90.000,E1 267.764} C_DIS
LIN {X 0.110,Y -458.437,Z 569.485,A 0.000,B 0.000,C 90.000,E1 267.306} C_DIS
LIN {X -0.032,Y -451.357,Z 569.483,A 0.000,B 0.000,C 90.000,E1 266.963} C_DIS
LIN {X -0.020,Y -444.037,Z 569.482,A 0.000,B 0.000,C 90.000,E1 266.674} C_DIS
LIN {X -0.031,Y -436.287,Z 569.480,A 0.000,B 0.000,C 90.000,E1 266.445} C_DIS
LIN {X -0.029,Y -428.282,Z 569.479,A 0.000,B 0.000,C 90.000,E1 266.274} C_DIS
LIN {X -0.086,Y -419.296,Z 569.479,A 0.000,B 0.000,C 90.000,E1 266.159} C_DIS
LIN {X -0.135,Y -410.069,Z 569.478,A 0.000,B 0.000,C 90.000,E1 266.102} C_DIS
LIN {X -0.211,Y -406.434,Z 569.478,A 0.000,B 0.000,C 90.000,E1 266.102} C_DIS
LIN {X 0.053,Y -180.922,Z 569.478,A 0.000,B 0.000,C 90.000,E1 266.045} C_DIS
LIN {X -0.084,Y -180.870,Z 569.472,A 0.000,B 0.000,C 90.000,E1 265.065} C_DIS
LIN {X -0.001,Y -178.931,Z 569.443,A 0.000,B 0.000,C 90.000,E1 259.803} C_DIS
LIN {X 0.038,Y -175.980,Z 569.415,A 0.000,B 0.000,C 90.000,E1 254.700} C_DIS
LIN {X -0.018,Y -175.472,Z 569.410,A 0.000,B 0.000,C 90.000,E1 253.866} C_DIS
LIN {X 0.039,Y -172.220,Z 569.387,A 0.000,B 0.000,C 90.000,E1 249.571} C_DIS
LIN {X 0.017,Y -171.697,Z 569.382,A 0.000,B 0.000,C 90.000,E1 248.720} C_DIS
LIN {X 0.093,Y -167.291,Z 569.353,A 0.000,B 0.000,C 90.000,E1 243.512} C_DIS
LIN {X 0.025,Y -166.667,Z 569.348,A 0.000,B 0.000,C 90.000,E1 242.666} C_DIS
LIN {X -0.059,Y -162.650,Z 569.324,A 0.000,B 0.000,C 90.000,E1 238.329} C_DIS
LIN {X 0.003,Y -161.339,Z 569.314,A 0.000,B 0.000,C 90.000,E1 236.548} C_DIS
LIN {X 0.046,Y -157.333,Z 569.290,A 0.000,B 0.000,C 90.000,E1 232.110} C_DIS
LIN {X -0.021,Y -155.317,Z 569.275,A 0.000,B 0.000,C 90.000,E1 229.461} C_DIS
LIN {X 0.017,Y -151.672,Z 569.250,A 0.000,B 0.000,C 90.000,E1 224.960} C_DIS
LIN {X -0.043,Y -150.537,Z 569.240,A 0.000,B 0.000,C 90.000,E1 223.176} C_DIS
LIN {X -0.009,Y -147.263,Z 569.215,A 0.000,B 0.000,C 90.000,E1 218.624} C_DIS
LIN {X 0.048,Y -145.289,Z 569.194,A 0.000,B 0.000,C 90.000,E1 214.945} C_DIS
LIN {X -0.044,Y -142.388,Z 569.164,A 0.000,B 0.000,C 90.000,E1 209.461} C_DIS
LIN {X 0.003,Y -141.367,Z 569.148,A 0.000,B 0.000,C 90.000,E1 206.668} C_DIS
LIN {X -0.019,Y -139.344,Z 569.112,A 0.000,B 0.000,C 90.000,E1 200.174} C_DIS
LIN {X -0.014,Y -139.015,Z 569.102,A 0.000,B 0.000,C 90.000,E1 198.308} C_DIS
LIN {X -0.018,Y -138.342,Z 569.055,A 0.000,B 0.000,C 90.000,E1 189.905} C_DIS
LIN {X 0.001,Y -139.395,Z 569.008,A 0.000,B 0.000,C 90.000,E1 181.489} C_DIS
LIN {X 0.055,Y -141.296,Z 568.972,A 0.000,B 0.000,C 90.000,E1 174.951} C_DIS
LIN {X 0.013,Y -142.659,Z 568.957,A 0.000,B 0.000,C 90.000,E1 172.186} C_DIS
LIN {X -0.037,Y -145.001,Z 568.931,A 0.000,B 0.000,C 90.000,E1 167.589} C_DIS
LIN {X -0.048,Y -147.629,Z 568.911,A 0.000,B 0.000,C 90.000,E1 163.921} C_DIS
LIN {X 0.030,Y -150.256,Z 568.890,A 0.000,B 0.000,C 90.000,E1 160.242} C_DIS
LIN {X 0.044,Y -153.655,Z 568.870,A 0.000,B 0.000,C 90.000,E1 156.613} C_DIS
LIN {X -0.039,Y -157.070,Z 568.850,A 0.000,B 0.000,C 90.000,E1 153.050} C_DIS
LIN {X 0.039,Y -161.202,Z 568.830,A 0.000,B 0.000,C 90.000,E1 149.459} C_DIS
LIN {X -0.012,Y -163.294,Z 568.821,A 0.000,B 0.000,C 90.000,E1 147.709} C_DIS
LIN {X -0.002,Y -167.740,Z 568.801,A 0.000,B 0.000,C 90.000,E1 144.196} C_DIS
LIN {X -0.090,Y -171.557,Z 568.787,A 0.000,B 0.000,C 90.000,E1 141.618} C_DIS
LIN {X -0.048,Y -176.503,Z 568.767,A 0.000,B 0.000,C 90.000,E1 138.162} C_DIS
LIN {X 0.077,Y -180.800,Z 568.753,A 0.000,B 0.000,C 90.000,E1 135.567} C_DIS
LIN {X 0.062,Y -186.208,Z 568.735,A 0.000,B 0.000,C 90.000,E1 132.204} C_DIS
LIN {X 0.019,Y -191.308,Z 568.719,A 0.000,B 0.000,C 90.000,E1 129.439} C_DIS
LIN {X -0.080,Y -191.619,Z 568.718,A 0.000,B 0.000,C 90.000,E1 129.277} C_DIS
LIN {X -0.151,Y -288.963,Z 568.718,A 0.000,B 0.000,C 90.000,E1 129.277} C_DIS
LIN {X 0.074,Y -290.816,Z 568.718,A 0.000,B 0.000,C 90.000,E1 129.197} C_DIS
LIN {X -0.064,Y -296.309,Z 568.716,A 0.000,B 0.000,C 90.000,E1 128.910} C_DIS
LIN {X 0.023,Y -299.501,Z 568.714,A 0.000,B 0.000,C 90.000,E1 128.543} C_DIS
LIN {X -0.075,Y -301.492,Z 568.712,A 0.000,B 0.000,C 90.000,E1 128.257} C_DIS
LIN {X 0.014,Y -303.053,Z 568.711,A 0.000,B 0.000,C 90.000,E1 127.935} C_DIS
LIN {X 0.024,Y -304.392,Z 568.709,A 0.000,B 0.000,C 90.000,E1 127.604} C_DIS
LIN {X -0.043,Y -307.266,Z 568.703,A 0.000,B 0.000,C 90.000,E1 126.629} C_DIS
LIN {X -0.024,Y -317.254,Z 568.685,A 0.000,B 0.000,C 90.000,E1 123.372} C_DIS
LIN {X 0.181,Y -327.556,Z 568.669,A 0.000,B 0.000,C 90.000,E1 120.463} C_DIS
LIN {X 0.187,Y -339.208,Z 568.654,A 0.000,B 0.000,C 90.000,E1 117.641} C_DIS
LIN {X 0.057,Y -352.311,Z 568.638,A 0.000,B 0.000,C 90.000,E1 114.899} C_DIS
LIN {X -0.074,Y -365.277,Z 568.625,A 0.000,B 0.000,C 90.000,E1 112.514} C_DIS
LIN {X 0.183,Y -379.577,Z 568.612,A 0.000,B 0.000,C 90.000,E1 110.120} C_DIS
LIN {X 0.196,Y -395.317,Z 568.599,A 0.000,B 0.000,C 90.000,E1 107.819} C_DIS
LIN {X -0.024,Y -412.611,Z 568.587,A 0.000,B 0.000,C 90.000,E1 105.607} C_DIS
LIN {X 0.066,Y -431.579,Z 568.575,A 0.000,B 0.000,C 90.000,E1 103.411} C_DIS
LIN {X -0.014,Y -451.674,Z 568.563,A 0.000,B 0.000,C 90.000,E1 101.366} C_DIS
LIN {X -0.086,Y -474.885,Z 568.551,A 0.000,B 0.000,C 90.000,E1 99.265} C_DIS
LIN {X -0.022,Y -476.916,Z 568.550,A 0.000,B 0.000,C 90.000,E1 99.029} C_DIS
LIN {X -0.032,Y -478.468,Z 568.549,A 0.000,B 0.000,C 90.000,E1 98.803} C_DIS
LIN {X -0.163,Y -479.772,Z 568.547,A 0.000,B 0.000,C 90.000,E1 98.568} C_DIS
LIN {X 0.180,Y -480.733,Z 568.546,A 0.000,B 0.000,C 90.000,E1 98.276} C_DIS
LIN {X -0.138,Y -481.804,Z 568.543,A 0.000,B 0.000,C 90.000,E1 97.814} C_DIS
LIN {X 0.028,Y -481.879,Z 568.541,A 0.000,B 0.000,C 90.000,E1 97.296} C_DIS
LIN {X 0.199,Y -480.970,Z 568.538,A 0.000,B 0.000,C 90.000,E1 96.777} C_DIS
LIN {X -0.105,Y -478.922,Z 568.535,A 0.000,B 0.000,C 90.000,E1 96.315} C_DIS
LIN {X 0.192,Y -477.339,Z 568.534,A 0.000,B 0.000,C 90.000,E1 96.030} C_DIS
LIN {X -0.008,Y -460.360,Z 568.521,A 0.000,B 0.000,C 90.000,E1 93.784} C_DIS
LIN {X 0.028,Y -450.214,Z 568.512,A 0.000,B 0.000,C 90.000,E1 92.236} C_DIS
LIN {X -0.012,Y -436.812,Z 568.499,A 0.000,B 0.000,C 90.000,E1 89.885} C_DIS
LIN {X -0.090,Y -429.144,Z 568.492,A 0.000,B 0.000,C 90.000,E1 88.568} C_DIS
LIN {X -0.024,Y -417.958,Z 568.482,A 0.000,B 0.000,C 90.000,E1 86.674} C_DIS
LIN {X -0.077,Y -405.408,Z 568.469,A 0.000,B 0.000,C 90.000,E1 84.489} C_DIS
LIN {X 0.076,Y -391.722,Z 568.455,A 0.000,B 0.000,C 90.000,E1 81.951} C_DIS
LIN {X -0.064,Y -379.746,Z 568.443,A 0.000,B 0.000,C 90.000,E1 79.690} C_DIS
LIN {X 0.020,Y -369.298,Z 568.431,A 0.000,B 0.000,C 90.000,E1 77.645} C_DIS
LIN {X -0.030,Y -356.520,Z 568.417,A 0.000,B 0.000,C 90.000,E1 74.991} C_DIS
LIN {X 0.116,Y -343.997,Z 568.400,A 0.000,B 0.000,C 90.000,E1 71.945} C_DIS
LIN {X -0.103,Y -332.899,Z 568.383,A 0.000,B 0.000,C 90.000,E1 68.901} C_DIS
LIN {X 0.083,Y -321.020,Z 568.362,A 0.000,B 0.000,C 90.000,E1 65.101} C_DIS
LIN {X -0.015,Y -313.508,Z 568.348,A 0.000,B 0.000,C 90.000,E1 62.564} C_DIS
LIN {X -0.139,Y -306.116,Z 568.333,A 0.000,B 0.000,C 90.000,E1 59.999} C_DIS
LIN {X -0.125,Y -298.848,Z 568.319,A 0.000,B 0.000,C 90.000,E1 57.375} C_DIS
LIN {X -0.056,Y -290.195,Z 568.300,A 0.000,B 0.000,C 90.000,E1 54.036} C_DIS
LIN {X 0.096,Y -285.200,Z 568.289,A 0.000,B 0.000,C 90.000,E1 51.984} C_DIS
LIN {X -0.122,Y -280.014,Z 568.278,A 0.000,B 0.000,C 90.000,E1 49.989} C_DIS
LIN {X -0.077,Y -276.325,Z 568.270,A 0.000,B 0.000,C 90.000,E1 48.609} C_DIS
LIN {X -0.095,Y -270.312,Z 568.258,A 0.000,B 0.000,C 90.000,E1 46.539} C_DIS
LIN {X 0.068,Y -264.757,Z 568.249,A 0.000,B 0.000,C 90.000,E1 44.757} C_DIS
LIN {X 0.022,Y -256.540,Z 568.235,A 0.000,B 0.000,C 90.000,E1 42.285} C_DIS
LIN {X 0.029,Y -245.293,Z 568.215,A 0.000,B 0.000,C 90.000,E1 38.669} C_DIS
LIN {X 0.034,Y -237.071,Z 568.198,A 0.000,B 0.000,C 90.000,E1 35.724} C_DIS
LIN {X -0.048,Y -229.539,Z 568.182,A 0.000,B 0.000,C 90.000,E1 32.752} C_DIS
LIN {X 0.139,Y -222.654,Z 568.165,A 0.000,B 0.000,C 90.000,E1 29.667} C_DIS
LIN {X 0.017,Y -216.580,Z 568.148,A 0.000,B 0.000,C 90.000,E1 26.616} C_DIS
LIN {X -0.010,Y -209.895,Z 568.126,A 0.000,B 0.000,C 90.000,E1 22.717} C_DIS
LIN {X -0.041,Y -206.694,Z 568.113,A 0.000,B 0.000,C 90.000,E1 20.355} C_DIS
LIN {X 0.013,Y -201.685,Z 568.086,A 0.000,B 0.000,C 90.000,E1 15.552} C_DIS
LIN {X 0.010,Y -198.013,Z 568.060,A 0.000,B 0.000,C 90.000,E1 10.715} C_DIS
LIN {X -0.099,Y -195.559,Z 568.023,A 0.000,B 0.000,C 90.000,E1 4.245} C_DIS
LIN {X 0.093,Y -197.180,Z 567.966,A 0.000,B 0.000,C 90.000,E1 353.799} C_DIS
LIN {X -0.081,Y -200.837,Z 567.934,A 0.000,B 0.000,C 90.000,E1 348.173} C_DIS
LIN {X 0.011,Y -205.377,Z 567.907,A 0.000,B 0.000,C 90.000,E1 343.323} C_DIS
LIN {X 0.023,Y -210.004,Z 567.885,A 0.000,B 0.000,C 90.000,E1 339.337} C_DIS
LIN {X -0.030,Y -215.296,Z 567.863,A 0.000,B 0.000,C 90.000,E1 335.409} C_DIS
LIN {X -0.031,Y -221.240,Z 567.842,A 0.000,B 0.000,C 90.000,E1 331.513} C_DIS
LIN {X -0.010,Y -227.823,Z 567.820,A 0.000,B 0.000,C 90.000,E1 327.661} C_DIS
LIN {X 0.007,Y -234.857,Z 567.799,A 0.000,B 0.000,C 90.000,E1 323.863} C_DIS
LIN {X 0.054,Y -242.424,Z 567.779,A 0.000,B 0.000,C 90.000,E1 320.114} C_DIS
LIN {X -0.055,Y -250.627,Z 567.758,A 0.000,B 0.000,C 90.000,E1 316.458} C_DIS
LIN {X -0.115,Y -260.151,Z 567.738,A 0.000,B 0.000,C 90.000,E1 312.852} C_DIS
LIN {X 0.029,Y -271.124,Z 567.718,A 0.000,B 0.000,C 90.000,E1 309.277} C_DIS
LIN {X 0.063,Y -283.664,Z 567.699,A 0.000,B 0.000,C 90.000,E1 305.804} C_DIS
LIN {X 0.081,Y -296.232,Z 567.682,A 0.000,B 0.000,C 90.000,E1 302.752} C_DIS
LIN {X 0.015,Y -311.305,Z 567.664,A 0.000,B 0.000,C 90.000,E1 299.461} C_DIS
LIN {X 0.000,Y -325.915,Z 567.648,A 0.000,B 0.000,C 90.000,E1 296.565} C_DIS
LIN {X -0.169,Y -342.041,Z 567.632,A 0.000,B 0.000,C 90.000,E1 293.770} C_DIS
LIN {X 0.067,Y -356.059,Z 567.620,A 0.000,B 0.000,C 90.000,E1 291.589} C_DIS
LIN {X 0.087,Y -375.840,Z 567.605,A 0.000,B 0.000,C 90.000,E1 288.906} C_DIS
LIN {X 0.056,Y -396.940,Z 567.591,A 0.000,B 0.000,C 90.000,E1 286.315} C_DIS
LIN {X 0.055,Y -413.760,Z 567.580,A 0.000,B 0.000,C 90.000,E1 284.356} C_DIS
LIN {X 0.160,Y -423.320,Z 567.574,A 0.000,B 0.000,C 90.000,E1 283.244} C_DIS
LIN {X 0.148,Y -434.738,Z 567.566,A 0.000,B 0.000,C 90.000,E1 281.895} C_DIS
LIN {X -0.126,Y -445.415,Z 567.559,A 0.000,B 0.000,C 90.000,E1 280.602} C_DIS
LIN {X -0.151,Y -453.359,Z 567.553,A 0.000,B 0.000,C 90.000,E1 279.557} C_DIS
LIN {X -0.081,Y -460.657,Z 567.547,A 0.000,B 0.000,C 90.000,E1 278.511} C_DIS
LIN {X 0.073,Y -467.355,Z 567.542,A 0.000,B 0.000,C 90.000,E1 277.466} C_DIS
LIN {X -0.070,Y -471.914,Z 567.537,A 0.000,B 0.000,C 90.000,E1 276.720} C_DIS
LIN {X -0.113,Y -476.002,Z 567.533,A 0.000,B 0.000,C 90.000,E1 275.967} C_DIS
LIN {X -0.177,Y -479.522,Z 567.529,A 0.000,B 0.000,C 90.000,E1 275.220} C_DIS
LIN {X -0.026,Y -481.534,Z 567.526,A 0.000,B 0.000,C 90.000,E1 274.702} C_DIS
LIN {X 0.094,Y -483.263,Z 567.523,A 0.000,B 0.000,C 90.000,E1 274.188} C_DIS
LIN {X -0.219,Y -484.698,Z 567.521,A 0.000,B 0.000,C 90.000,E1 273.726} C_DIS
LIN {X -0.071,Y -485.833,Z 567.518,A 0.000,B 0.000,C 90.000,E1 273.212} C_DIS
LIN {X 0.114,Y -486.614,Z 567.515,A 0.000,B 0.000,C 90.000,E1 272.694} C_DIS
LIN {X -0.206,Y -487.059,Z 567.512,A 0.000,B 0.000,C 90.000,E1 272.236} C_DIS
LIN {X -0.016,Y -487.029,Z 567.510,A 0.000,B 0.000,C 90.000,E1 271.718} C_DIS
LIN {X 0.159,Y -486.567,Z 567.507,A 0.000,B 0.000,C 90.000,E1 271.203} C_DIS
LIN {X -0.150,Y -485.593,Z 567.504,A 0.000,B 0.000,C 90.000,E1 270.745} C_DIS
LIN {X 0.024,Y -484.044,Z 567.501,A 0.000,B 0.000,C 90.000,E1 270.229} C_DIS
LIN {X 0.192,Y -481.882,Z 567.499,A 0.000,B 0.000,C 90.000,E1 269.714} C_DIS
LIN {X -0.130,Y -478.993,Z 567.496,A 0.000,B 0.000,C 90.000,E1 269.255} C_DIS
LIN {X 0.007,Y -475.306,Z 567.493,A 0.000,B 0.000,C 90.000,E1 268.740} C_DIS
LIN {X 0.122,Y -470.572,Z 567.490,A 0.000,B 0.000,C 90.000,E1 268.224} C_DIS
LIN {X -0.013,Y -467.861,Z 567.489,A 0.000,B 0.000,C 90.000,E1 267.993} C_DIS
LIN {X -0.160,Y -464.792,Z 567.487,A 0.000,B 0.000,C 90.000,E1 267.764} C_DIS
LIN {X -0.050,Y -461.745,Z 567.486,A 0.000,B 0.000,C 90.000,E1 267.535} C_DIS
LIN {X 0.058,Y -458.291,Z 567.485,A 0.000,B 0.000,C 90.000,E1 267.306} C_DIS
LIN {X -0.050,Y -451.263,Z 567.483,A 0.000,B 0.000,C 90.000,E1 266.963} C_DIS
LIN {X -0.025,Y -443.985,Z 567.482,A 0.000,B 0.000,C 90.000,E1 266.674} C_DIS
LIN {X -0.026,Y -436.380,Z 567.480,A 0.000,B 0.000,C 90.000,E1 266.445} C_DIS
LIN {X -0.055,Y -428.188,Z 567.479,A 0.000,B 0.000,C 90.000,E1 266.274} C_DIS
LIN {X -0.127,Y -419.064,Z 567.479,A 0.000,B 0.000,C 90.000,E1 266.159} C_DIS
LIN {X -0.173,Y -409.130,Z 567.478,A 0.000,B 0.000,C 90.000,E1 266.102} C_DIS
LIN {X 0.070,Y -180.923,Z 567.478,A 0.000,B 0.000,C 90.000,E1 266.045} C_DIS
LIN {X -0.068,Y -180.871,Z 567.472,A 0.000,B 0.000,C 90.000,E1 265.065} C_DIS
LIN {X 0.015,Y -178.934,Z 567.443,A 0.000,B 0.000,C 90.000,E1 259.803} C_DIS
LIN {X 0.053,Y -175.982,Z 567.415,A 0.000,B 0.000,C 90.000,E1 254.700} C_DIS
LIN {X -0.002,Y -175.476,Z 567.410,A 0.000,B 0.000,C 90.000,E1 253.866} C_DIS
LIN {X 0.054,Y -172.224,Z 567.387,A 0.000,B 0.000,C 90.000,E1 249.571} C_DIS
LIN {X 0.032,Y -171.699,Z 567.382,A 0.000,B 0.000,C 90.000,E1 248.720} C_DIS
LIN {X -0.043,Y -167.294,Z 567.353,A 0.000,B 0.000,C 90.000,E1 243.563} C_DIS
LIN {X 0.039,Y -166.672,Z 567.348,A 0.000,B 0.000,C 90.000,E1 242.666} C_DIS
LIN {X -0.045,Y -162.654,Z 567.324,A 0.000,B 0.000,C 90.000,E1 238.329} C_DIS
LIN {X 0.017,Y -161.343,Z 567.314,A 0.000,B 0.000,C 90.000,E1 236.548} C_DIS
LIN {X 0.060,Y -157.337,Z 567.290,A 0.000,B 0.000,C 90.000,E1 232.110} C_DIS
LIN {X -0.007,Y -155.322,Z 567.275,A 0.000,B 0.000,C 90.000,E1 229.461} C_DIS
LIN {X -0.077,Y -151.675,Z 567.250,A 0.000,B 0.000,C 90.000,E1 225.000} C_DIS
LIN {X -0.029,Y -150.540,Z 567.240,A 0.000,B 0.000,C 90.000,E1 223.176} C_DIS
LIN {X 0.004,Y -147.265,Z 567.215,A 0.000,B 0.000,C 90.000,E1 218.624} C_DIS
LIN {X -0.023,Y -145.293,Z 567.194,A 0.000,B 0.000,C 90.000,E1 214.978} C_DIS
LIN {X -0.030,Y -142.390,Z 567.164,A 0.000,B 0.000,C 90.000,E1 209.461} C_DIS
LIN {X 0.016,Y -141.369,Z 567.148,A 0.000,B 0.000,C 90.000,E1 206.668} C_DIS
LIN {X -0.005,Y -139.345,Z 567.112,A 0.000,B 0.000,C 90.000,E1 200.174} C_DIS
LIN {X -0.001,Y -139.017,Z 567.102,A 0.000,B 0.000,C 90.000,E1 198.308} C_DIS
LIN {X -0.005,Y -138.342,Z 567.055,A 0.000,B 0.000,C 90.000,E1 189.905} C_DIS
LIN {X 0.015,Y -139.393,Z 567.008,A 0.000,B 0.000,C 90.000,E1 181.489} C_DIS
LIN {X 0.069,Y -141.294,Z 566.972,A 0.000,B 0.000,C 90.000,E1 174.951} C_DIS
LIN {X 0.026,Y -142.656,Z 566.957,A 0.000,B 0.000,C 90.000,E1 172.186} C_DIS
LIN {X -0.024,Y -144.998,Z 566.931,A 0.000,B 0.000,C 90.000,E1 167.589} C_DIS
LIN {X -0.034,Y -147.626,Z 566.911,A 0.000,B 0.000,C 90.000,E1 163.921} C_DIS
LIN {X 0.044,Y -150.253,Z 566.890,A 0.000,B 0.000,C 90.000,E1 160.242} C_DIS
LIN {X 0.059,Y -153.650,Z 566.870,A 0.000,B 0.000,C 90.000,E1 156.613} C_DIS
LIN {X -0.025,Y -157.065,Z 566.850,A 0.000,B 0.000,C 90.000,E1 153.050} C_DIS
LIN {X 0.054,Y -161.196,Z 566.830,A 0.000,B 0.000,C 90.000,E1 149.459} C_DIS
LIN {X 0.003,Y -163.288,Z 566.821,A 0.000,B 0.000,C 90.000,E1 147.709} C_DIS
LIN {X 0.012,Y -167.732,Z 566.801,A 0.000,B 0.000,C 90.000,E1 144.196} C_DIS
LIN {X -0.075,Y -171.551,Z 566.787,A 0.000,B 0.000,C 90.000,E1 141.618} C_DIS
LIN {X -0.033,Y -176.495,Z 566.768,A 0.000,B 0.000,C 90.000,E1 138.162} C_DIS
LIN {X 0.092,Y -180.792,Z 566.753,A 0.000,B 0.000,C 90.000,E1 135.567} C_DIS
LIN {X -0.048,Y -186.200,Z 566.735,A 0.000,B 0.000,C 90.000,E1 132.243} C_DIS
LIN {X 0.081,Y -191.408,Z 566.719,A 0.000,B 0.000,C 90.000,E1 129.358} C_DIS
LIN {X -0.005,Y -191.642,Z 566.718,A 0.000,B 0.000,C 90.000,E1 129.241} C_DIS
LIN {X 0.186,Y -288.776,Z 566.718,A 0.000,B 0.000,C 90.000,E1 129.197} C_DIS
LIN {X 0.096,Y -290.024,Z 566.718,A 0.000,B 0.000,C 90.000,E1 129.197} C_DIS
LIN {X -0.064,Y -293.930,Z 566.717,A 0.000,B 0.000,C 90.000,E1 129.072} C_DIS
LIN {X -0.039,Y -296.092,Z 566.716,A 0.000,B 0.000,C 90.000,E1 128.910} C_DIS
LIN {X 0.033,Y -299.976,Z 566.714,A 0.000,B 0.000,C 90.000,E1 128.463} C_DIS
LIN {X -0.086,Y -301.885,Z 566.712,A 0.000,B 0.000,C 90.000,E1 128.177} C_DIS
LIN {X -0.018,Y -303.388,Z 566.710,A 0.000,B 0.000,C 90.000,E1 127.855} C_DIS
LIN {X -0.007,Y -304.661,Z 566.708,A 0.000,B 0.000,C 90.000,E1 127.523} C_DIS
LIN {X 0.157,Y -316.441,Z 566.687,A 0.000,B 0.000,C 90.000,E1 123.579} C_DIS
LIN {X 0.061,Y -326.637,Z 566.671,A 0.000,B 0.000,C 90.000,E1 120.718} C_DIS
LIN {X 0.035,Y -338.172,Z 566.655,A 0.000,B 0.000,C 90.000,E1 117.897} C_DIS
LIN {X -0.135,Y -351.155,Z 566.640,A 0.000,B 0.000,C 90.000,E1 115.155} C_DIS
LIN {X 0.037,Y -364.001,Z 566.626,A 0.000,B 0.000,C 90.000,E1 112.717} C_DIS
LIN {X 0.053,Y -378.173,Z 566.613,A 0.000,B 0.000,C 90.000,E1 110.355} C_DIS
LIN {X 0.019,Y -393.776,Z 566.600,A 0.000,B 0.000,C 90.000,E1 108.055} C_DIS
LIN {X 0.144,Y -410.921,Z 566.588,A 0.000,B 0.000,C 90.000,E1 105.788} C_DIS
LIN {X 0.197,Y -429.737,Z 566.576,A 0.000,B 0.000,C 90.000,E1 103.592} C_DIS
LIN {X 0.086,Y -449.778,Z 566.564,A 0.000,B 0.000,C 90.000,E1 101.535} C_DIS
LIN {X -0.193,Y -470.376,Z 566.554,A 0.000,B 0.000,C 90.000,E1 99.670} C_DIS
LIN {X -0.099,Y -475.458,Z 566.551,A 0.000,B 0.000,C 90.000,E1 99.208} C_DIS
LIN {X -0.070,Y -477.410,Z 566.550,A 0.000,B 0.000,C 90.000,E1 98.973} C_DIS
LIN {X -0.115,Y -478.900,Z 566.549,A 0.000,B 0.000,C 90.000,E1 98.746} C_DIS
LIN {X 0.232,Y -480.125,Z 566.547,A 0.000,B 0.000,C 90.000,E1 98.454} C_DIS
LIN {X 0.101,Y -481.020,Z 566.546,A 0.000,B 0.000,C 90.000,E1 98.219} C_DIS
LIN {X -0.214,Y -481.980,Z 566.543,A 0.000,B 0.000,C 90.000,E1 97.757} C_DIS
LIN {X -0.047,Y -481.951,Z 566.540,A 0.000,B 0.000,C 90.000,E1 97.239} C_DIS
LIN {X 0.127,Y -480.932,Z 566.537,A 0.000,B 0.000,C 90.000,E1 96.720} C_DIS
LIN {X 0.003,Y -480.005,Z 566.536,A 0.000,B 0.000,C 90.000,E1 96.486} C_DIS
LIN {X -0.175,Y -478.744,Z 566.535,A 0.000,B 0.000,C 90.000,E1 96.258} C_DIS
LIN {X -0.013,Y -475.134,Z 566.532,A 0.000,B 0.000,C 90.000,E1 95.739} C_DIS
LIN {X -0.087,Y -460.064,Z 566.521,A 0.000,B 0.000,C 90.000,E1 93.726} C_DIS
LIN {X 0.181,Y -451.509,Z 566.513,A 0.000,B 0.000,C 90.000,E1 92.407} C_DIS
LIN {X -0.097,Y -436.540,Z 566.499,A 0.000,B 0.000,C 90.000,E1 89.828} C_DIS
LIN {X -0.178,Y -428.809,Z 566.492,A 0.000,B 0.000,C 90.000,E1 88.511} C_DIS
LIN {X -0.012,Y -416.037,Z 566.480,A 0.000,B 0.000,C 90.000,E1 86.331} C_DIS
LIN {X -0.028,Y -402.004,Z 566.466,A 0.000,B 0.000,C 90.000,E1 83.856} C_DIS
LIN {X 0.026,Y -389.881,Z 566.453,A 0.000,B 0.000,C 90.000,E1 81.602} C_DIS
LIN {X -0.178,Y -379.393,Z 566.442,A 0.000,B 0.000,C 90.000,E1 79.634} C_DIS
LIN {X -0.101,Y -368.909,Z 566.431,A 0.000,B 0.000,C 90.000,E1 77.589} C_DIS
LIN {X -0.119,Y -357.472,Z 566.418,A 0.000,B 0.000,C 90.000,E1 75.227} C_DIS
LIN {X 0.045,Y -346.037,Z 566.403,A 0.000,B 0.000,C 90.000,E1 72.489} C_DIS
LIN {X -0.119,Y -334.746,Z 566.386,A 0.000,B 0.000,C 90.000,E1 69.444} C_DIS
LIN {X 0.015,Y -322.701,Z 566.365,A 0.000,B 0.000,C 90.000,E1 65.665} C_DIS
LIN {X -0.037,Y -315.141,Z 566.351,A 0.000,B 0.000,C 90.000,E1 63.127} C_DIS
LIN {X 0.004,Y -307.742,Z 566.336,A 0.000,B 0.000,C 90.000,E1 60.539} C_DIS
LIN {X 0.051,Y -300.429,Z 566.322,A 0.000,B 0.000,C 90.000,E1 57.916} C_DIS
LIN {X -0.001,Y -291.670,Z 566.303,A 0.000,B 0.000,C 90.000,E1 54.609} C_DIS
LIN {X 0.066,Y -284.981,Z 566.288,A 0.000,B 0.000,C 90.000,E1 51.904} C_DIS
LIN {X -0.155,Y -279.768,Z 566.277,A 0.000,B 0.000,C 90.000,E1 49.908} C_DIS
LIN {X 0.095,Y -276.049,Z 566.269,A 0.000,B 0.000,C 90.000,E1 48.485} C_DIS
LIN {X -0.112,Y -272.048,Z 566.262,A 0.000,B 0.000,C 90.000,E1 47.148} C_DIS
LIN {X 0.019,Y -267.770,Z 566.254,A 0.000,B 0.000,C 90.000,E1 45.729} C_DIS
LIN {X 0.135,Y -262.026,Z 566.244,A 0.000,B 0.000,C 90.000,E1 43.947} C_DIS
LIN {X -0.090,Y -251.573,Z 566.226,A 0.000,B 0.000,C 90.000,E1 40.782} C_DIS
LIN {X -0.023,Y -242.801,Z 566.210,A 0.000,B 0.000,C 90.000,E1 37.855} C_DIS
LIN {X -0.026,Y -234.804,Z 566.194,A 0.000,B 0.000,C 90.000,E1 34.898} C_DIS
LIN {X 0.032,Y -227.424,Z 566.177,A 0.000,B 0.000,C 90.000,E1 31.878} C_DIS
LIN {X 0.052,Y -220.773,Z 566.160,A 0.000,B 0.000,C 90.000,E1 28.821} C_DIS
LIN {X 0.081,Y -214.898,Z 566.143,A 0.000,B 0.000,C 90.000,E1 25.720} C_DIS
LIN {X 0.074,Y -209.693,Z 566.126,A 0.000,B 0.000,C 90.000,E1 22.589} C_DIS
LIN {X -0.037,Y -206.555,Z 566.112,A 0.000,B 0.000,C 90.000,E1 20.248} C_DIS
LIN {X 0.076,Y -201.537,Z 566.086,A 0.000,B 0.000,C 90.000,E1 15.426} C_DIS
LIN {X 0.022,Y -197.908,Z 566.059,A 0.000,B 0.000,C 90.000,E1 10.602} C_DIS
LIN {X 0.071,Y -195.398,Z 566.018,A 0.000,B 0.000,C 90.000,E1 3.269} C_DIS
LIN {X 0.092,Y -197.161,Z 565.966,A 0.000,B 0.000,C 90.000,E1 353.799} C_DIS
LIN {X -0.082,Y -200.831,Z 565.934,A 0.000,B 0.000,C 90.000,E1 348.173} C_DIS
LIN {X 0.009,Y -205.364,Z 565.907,A 0.000,B 0.000,C 90.000,E1 343.323} C_DIS
LIN {X 0.020,Y -209.974,Z 565.885,A 0.000,B 0.000,C 90.000,E1 339.337} C_DIS
LIN {X -0.032,Y -215.286,Z 565.863,A 0.000,B 0.000,C 90.000,E1 335.409} C_DIS
LIN {X -0.035,Y -221.223,Z 565.842,A 0.000,B 0.000,C 90.000,E1 331.513} C_DIS
LIN {X -0.014,Y -227.791,Z 565.820,A 0.000,B 0.000,C 90.000,E1 327.661} C_DIS
LIN {X 0.001,Y -234.810,Z 565.799,A 0.000,B 0.000,C 90.000,E1 323.863} C_DIS
LIN {X 0.047,Y -242.392,Z 565.778,A 0.000,B 0.000,C 90.000,E1 320.114} C_DIS
LIN {X -0.063,Y -250.598,Z 565.758,A 0.000,B 0.000,C 90.000,E1 316.458} C_DIS
LIN {X -0.124,Y -260.158,Z 565.738,A 0.000,B 0.000,C 90.000,E1 312.852} C_DIS
LIN {X 0.020,Y -271.130,Z 565.718,A 0.000,B 0.000,C 90.000,E1 309.277} C_DIS
LIN {X -0.060,Y -282.330,Z 565.701,A 0.000,B 0.000,C 90.000,E1 306.171} C_DIS
LIN {X -0.071,Y -293.279,Z 565.686,A 0.000,B 0.000,C 90.000,E1 303.452} C_DIS
LIN {X -0.106,Y -306.576,Z 565.669,A 0.000,B 0.000,C 90.000,E1 300.463} C_DIS
LIN {X -0.033,Y -322.497,Z 565.651,A 0.000,B 0.000,C 90.000,E1 297.206} C_DIS
LIN {X 0.148,Y -338.185,Z 565.635,A 0.000,B 0.000,C 90.000,E1 294.335} C_DIS
LIN {X -0.016,Y -351.843,Z 565.623,A 0.000,B 0.000,C 90.000,E1 292.206} C_DIS
LIN {X -0.080,Y -369.049,Z 565.610,A 0.000,B 0.000,C 90.000,E1 289.812} C_DIS
LIN {X 0.067,Y -389.805,Z 565.595,A 0.000,B 0.000,C 90.000,E1 287.166} C_DIS
LIN {X 0.023,Y -406.543,Z 565.584,A 0.000,B 0.000,C 90.000,E1 285.190} C_DIS
LIN {X 0.015,Y -418.474,Z 565.577,A 0.000,B 0.000,C 90.000,E1 283.828} C_DIS
LIN {X -0.076,Y -430.139,Z 565.569,A 0.000,B 0.000,C 90.000,E1 282.479} C_DIS
LIN {X -0.193,Y -438.987,Z 565.563,A 0.000,B 0.000,C 90.000,E1 281.422} C_DIS
LIN {X 0.227,Y -447.426,Z 565.557,A 0.000,B 0.000,C 90.000,E1 280.310} C_DIS
LIN {X 0.233,Y -455.195,Z 565.552,A 0.000,B 0.000,C 90.000,E1 279.265} C_DIS
LIN {X -0.129,Y -462.397,Z 565.546,A 0.000,B 0.000,C 90.000,E1 278.276} C_DIS
LIN {X -0.019,Y -468.919,Z 565.540,A 0.000,B 0.000,C 90.000,E1 277.239} C_DIS
LIN {X -0.087,Y -473.289,Z 565.536,A 0.000,B 0.000,C 90.000,E1 276.486} C_DIS
LIN {X -0.175,Y -477.213,Z 565.532,A 0.000,B 0.000,C 90.000,E1 275.739} C_DIS
LIN {X -0.037,Y -479.500,Z 565.529,A 0.000,B 0.000,C 90.000,E1 275.220} C_DIS
LIN {X 0.114,Y -481.524,Z 565.526,A 0.000,B 0.000,C 90.000,E1 274.702} C_DIS
LIN {X -0.247,Y -483.260,Z 565.523,A 0.000,B 0.000,C 90.000,E1 274.245} C_DIS
LIN {X -0.079,Y -484.679,Z 565.521,A 0.000,B 0.000,C 90.000,E1 273.726} C_DIS
LIN {X 0.070,Y -485.792,Z 565.518,A 0.000,B 0.000,C 90.000,E1 273.212} C_DIS
LIN {X -0.231,Y -486.602,Z 565.515,A 0.000,B 0.000,C 90.000,E1 272.751} C_DIS
LIN {X -0.064,Y -487.021,Z 565.512,A 0.000,B 0.000,C 90.000,E1 272.236} C_DIS
LIN {X 0.125,Y -487.017,Z 565.510,A 0.000,B 0.000,C 90.000,E1 271.718} C_DIS
LIN {X -0.186,Y -486.544,Z 565.507,A 0.000,B 0.000,C 90.000,E1 271.260} C_DIS
LIN {X -0.010,Y -485.586,Z 565.504,A 0.000,B 0.000,C 90.000,E1 270.745} C_DIS
LIN {X 0.165,Y -484.076,Z 565.501,A 0.000,B 0.000,C 90.000,E1 270.229} C_DIS
LIN {X -0.150,Y -481.936,Z 565.499,A 0.000,B 0.000,C 90.000,E1 269.771} C_DIS
LIN {X 0.009,Y -479.084,Z 565.496,A 0.000,B 0.000,C 90.000,E1 269.255} C_DIS
LIN {X 0.145,Y -475.402,Z 565.493,A 0.000,B 0.000,C 90.000,E1 268.740} C_DIS
LIN {X -0.034,Y -473.214,Z 565.492,A 0.000,B 0.000,C 90.000,E1 268.511} C_DIS
LIN {X 0.117,Y -468.025,Z 565.489,A 0.000,B 0.000,C 90.000,E1 267.993} C_DIS
LIN {X -0.039,Y -464.950,Z 565.488,A 0.000,B 0.000,C 90.000,E1 267.764} C_DIS
LIN {X 0.069,Y -461.920,Z 565.486,A 0.000,B 0.000,C 90.000,E1 267.535} C_DIS
LIN {X 0.113,Y -455.231,Z 565.484,A 0.000,B 0.000,C 90.000,E1 267.135} C_DIS
LIN {X -0.151,Y -448.128,Z 565.482,A 0.000,B 0.000,C 90.000,E1 266.846} C_DIS
LIN {X 0.060,Y -440.815,Z 565.481,A 0.000,B 0.000,C 90.000,E1 266.560} C_DIS
LIN {X -0.199,Y -432.947,Z 565.480,A 0.000,B 0.000,C 90.000,E1 266.388} C_DIS
LIN {X -0.089,Y -424.474,Z 565.479,A 0.000,B 0.000,C 90.000,E1 266.216} C_DIS
LIN {X -0.053,Y -413.519,Z 565.478,A 0.000,B 0.000,C 90.000,E1 266.102} C_DIS
LIN {X -0.204,Y -408.600,Z 565.478,A 0.000,B 0.000,C 90.000,E1 266.102} C_DIS
LIN {X 0.056,Y -180.923,Z 565.478,A 0.000,B 0.000,C 90.000,E1 266.045} C_DIS
LIN {X -0.082,Y -180.871,Z 565.472,A 0.000,B 0.000,C 90.000,E1 265.065} C_DIS
LIN {X 0.001,Y -178.932,Z 565.443,A 0.000,B 0.000,C 90.000,E1 259.803} C_DIS
LIN {X 0.039,Y -175.980,Z 565.415,A 0.000,B 0.000,C 90.000,E1 254.700} C_DIS
LIN {X -0.016,Y -175.473,Z 565.410,A 0.000,B 0.000,C 90.000,E1 253.866} C_DIS
LIN {X 0.040,Y -172.220,Z 565.387,A 0.000,B 0.000,C 90.000,E1 249.571} C_DIS
LIN {X 0.018,Y -171.696,Z 565.382,A 0.000,B 0.000,C 90.000,E1 248.720} C_DIS
LIN {X 0.094,Y -167.291,Z 565.353,A 0.000,B 0.000,C 90.000,E1 243.512} C_DIS
LIN {X 0.027,Y -166.668,Z 565.348,A 0.000,B 0.000,C 90.000,E1 242.666} C_DIS
LIN {X -0.058,Y -162.650,Z 565.324,A 0.000,B 0.000,C 90.000,E1 238.329} C_DIS
LIN {X 0.004,Y -161.339,Z 565.314,A 0.000,B 0.000,C 90.000,E1 236.548} C_DIS
LIN {X 0.047,Y -157.334,Z 565.290,A 0.000,B 0.000,C 90.000,E1 232.110} C_DIS
LIN {X -0.021,Y -155.318,Z 565.275,A 0.000,B 0.000,C 90.000,E1 229.461} C_DIS
LIN {X 0.018,Y -151.672,Z 565.250,A 0.000,B 0.000,C 90.000,E1 224.960} C_DIS
LIN {X -0.041,Y -150.537,Z 565.240,A 0.000,B 0.000,C 90.000,E1 223.176} C_DIS
LIN {X -0.008,Y -147.262,Z 565.215,A 0.000,B 0.000,C 90.000,E1 218.624} C_DIS
LIN {X 0.048,Y -145.289,Z 565.194,A 0.000,B 0.000,C 90.000,E1 214.945} C_DIS
LIN {X -0.042,Y -142.388,Z 565.164,A 0.000,B 0.000,C 90.000,E1 209.461} C_DIS
LIN {X 0.004,Y -141.367,Z 565.148,A 0.000,B 0.000,C 90.000,E1 206.668} C_DIS
LIN {X -0.018,Y -139.345,Z 565.112,A 0.000,B 0.000,C 90.000,E1 200.174} C_DIS
LIN {X -0.012,Y -139.015,Z 565.102,A 0.000,B 0.000,C 90.000,E1 198.308} C_DIS
LIN {X -0.017,Y -138.342,Z 565.055,A 0.000,B 0.000,C 90.000,E1 189.905} C_DIS
LIN {X 0.003,Y -139.395,Z 565.008,A 0.000,B 0.000,C 90.000,E1 181.489} C_DIS
LIN {X 0.057,Y -141.296,Z 564.972,A 0.000,B 0.000,C 90.000,E1 174.951} C_DIS
LIN {X 0.014,Y -142.659,Z 564.957,A 0.000,B 0.000,C 90.000,E1 172.186} C_DIS
LIN {X -0.035,Y -145.001,Z 564.931,A 0.000,B 0.000,C 90.000,E1 167.589} C_DIS
LIN {X -0.046,Y -147.628,Z 564.911,A 0.000,B 0.000,C 90.000,E1 163.921} C_DIS
LIN {X 0.032,Y -150.257,Z 564.890,A 0.000,B 0.000,C 90.000,E1 160.242} C_DIS
LIN {X 0.045,Y -153.654,Z 564.870,A 0.000,B 0.000,C 90.000,E1 156.613} C_DIS
LIN {X -0.038,Y -157.069,Z 564.850,A 0.000,B 0.000,C 90.000,E1 153.050} C_DIS
LIN {X 0.041,Y -161.201,Z 564.830,A 0.000,B 0.000,C 90.000,E1 149.459} C_DIS
LIN {X -0.010,Y -163.293,Z 564.821,A 0.000,B 0.000,C 90.000,E1 147.709} C_DIS
LIN {X 0.000,Y -167.739,Z 564.801,A 0.000,B 0.000,C 90.000,E1 144.196} C_DIS
LIN {X -0.088,Y -171.557,Z 564.787,A 0.000,B 0.000,C 90.000,E1 141.618} C_DIS
LIN {X -0.047,Y -176.501,Z 564.767,A 0.000,B 0.000,C 90.000,E1 138.162} C_DIS
LIN {X 0.077,Y -180.799,Z 564.753,A 0.000,B 0.000,C 90.000,E1 135.567} C_DIS
LIN {X 0.064,Y -186.207,Z 564.735,A 0.000,B 0.000,C 90.000,E1 132.204} C_DIS
LIN {X 0.019,Y -191.308,Z 564.719,A 0.000,B 0.000,C 90.000,E1 129.439} C_DIS
LIN {X 0.088,Y -191.669,Z 564.718,A 0.000,B 0.000,C 90.000,E1 129.197} C_DIS
LIN {X 0.101,Y -288.781,Z 564.718,A 0.000,B 0.000,C 90.000,E1 129.197} C_DIS
LIN {X 0.099,Y -293.747,Z 564.717,A 0.000,B 0.000,C 90.000,E1 129.036} C_DIS
LIN {X -0.061,Y -295.967,Z 564.716,A 0.000,B 0.000,C 90.000,E1 128.910} C_DIS
LIN {X 0.067,Y -299.836,Z 564.714,A 0.000,B 0.000,C 90.000,E1 128.463} C_DIS
LIN {X -0.026,Y -301.756,Z 564.712,A 0.000,B 0.000,C 90.000,E1 128.177} C_DIS
LIN {X -0.119,Y -303.270,Z 564.710,A 0.000,B 0.000,C 90.000,E1 127.890} C_DIS
LIN {X 0.078,Y -304.573,Z 564.709,A 0.000,B 0.000,C 90.000,E1 127.523} C_DIS
LIN {X 0.181,Y -315.316,Z 564.689,A 0.000,B 0.000,C 90.000,E1 123.913} C_DIS
LIN {X 0.054,Y -325.361,Z 564.673,A 0.000,B 0.000,C 90.000,E1 121.052} C_DIS
LIN {X -0.012,Y -336.737,Z 564.657,A 0.000,B 0.000,C 90.000,E1 118.231} C_DIS
LIN {X -0.064,Y -349.542,Z 564.641,A 0.000,B 0.000,C 90.000,E1 115.463} C_DIS
LIN {X 0.064,Y -362.221,Z 564.628,A 0.000,B 0.000,C 90.000,E1 113.025} C_DIS
LIN {X 0.038,Y -376.213,Z 564.615,A 0.000,B 0.000,C 90.000,E1 110.663} C_DIS
LIN {X -0.044,Y -391.622,Z 564.602,A 0.000,B 0.000,C 90.000,E1 108.362} C_DIS
LIN {X 0.143,Y -408.558,Z 564.589,A 0.000,B 0.000,C 90.000,E1 106.079} C_DIS
LIN {X 0.131,Y -427.146,Z 564.577,A 0.000,B 0.000,C 90.000,E1 103.883} C_DIS
LIN {X -0.151,Y -447.084,Z 564.566,A 0.000,B 0.000,C 90.000,E1 101.827} C_DIS
LIN {X -0.156,Y -467.613,Z 564.555,A 0.000,B 0.000,C 90.000,E1 99.905} C_DIS
LIN {X -0.018,Y -475.355,Z 564.551,A 0.000,B 0.000,C 90.000,E1 99.208} C_DIS
LIN {X 0.033,Y -477.344,Z 564.550,A 0.000,B 0.000,C 90.000,E1 98.973} C_DIS
LIN {X 0.009,Y -478.865,Z 564.549,A 0.000,B 0.000,C 90.000,E1 98.746} C_DIS
LIN {X -0.120,Y -480.130,Z 564.547,A 0.000,B 0.000,C 90.000,E1 98.511} C_DIS
LIN {X 0.225,Y -481.058,Z 564.546,A 0.000,B 0.000,C 90.000,E1 98.219} C_DIS
LIN {X -0.091,Y -482.075,Z 564.543,A 0.000,B 0.000,C 90.000,E1 97.757} C_DIS
LIN {X 0.077,Y -482.100,Z 564.540,A 0.000,B 0.000,C 90.000,E1 97.239} C_DIS
LIN {X -0.226,Y -481.138,Z 564.537,A 0.000,B 0.000,C 90.000,E1 96.777} C_DIS
LIN {X -0.051,Y -479.023,Z 564.535,A 0.000,B 0.000,C 90.000,E1 96.258} C_DIS
LIN {X -0.179,Y -477.391,Z 564.533,A 0.000,B 0.000,C 90.000,E1 96.024} C_DIS
LIN {X 0.047,Y -460.347,Z 564.521,A 0.000,B 0.000,C 90.000,E1 93.726} C_DIS
LIN {X -0.137,Y -451.767,Z 564.514,A 0.000,B 0.000,C 90.000,E1 92.465} C_DIS
LIN {X 0.039,Y -436.748,Z 564.499,A 0.000,B 0.000,C 90.000,E1 89.828} C_DIS
LIN {X -0.041,Y -428.991,Z 564.492,A 0.000,B 0.000,C 90.000,E1 88.511} C_DIS
LIN {X 0.125,Y -416.209,Z 564.480,A 0.000,B 0.000,C 90.000,E1 86.331} C_DIS
LIN {X 0.110,Y -402.189,Z 564.466,A 0.000,B 0.000,C 90.000,E1 83.856} C_DIS
LIN {X 0.163,Y -390.045,Z 564.453,A 0.000,B 0.000,C 90.000,E1 81.602} C_DIS
LIN {X -0.041,Y -379.519,Z 564.442,A 0.000,B 0.000,C 90.000,E1 79.634} C_DIS
LIN {X 0.035,Y -368.999,Z 564.431,A 0.000,B 0.000,C 90.000,E1 77.589} C_DIS
LIN {X 0.014,Y -357.530,Z 564.418,A 0.000,B 0.000,C 90.000,E1 75.227} C_DIS
LIN {X -0.154,Y -346.109,Z 564.403,A 0.000,B 0.000,C 90.000,E1 72.543} C_DIS
LIN {X 0.010,Y -334.820,Z 564.386,A 0.000,B 0.000,C 90.000,E1 69.444} C_DIS
LIN {X 0.141,Y -322.778,Z 564.365,A 0.000,B 0.000,C 90.000,E1 65.665} C_DIS
LIN {X 0.089,Y -315.223,Z 564.351,A 0.000,B 0.000,C 90.000,E1 63.127} C_DIS
LIN {X -0.140,Y -307.824,Z 564.336,A 0.000,B 0.000,C 90.000,E1 60.589} C_DIS
LIN {X 0.015,Y -300.521,Z 564.322,A 0.000,B 0.000,C 90.000,E1 57.946} C_DIS
LIN {X 0.121,Y -291.728,Z 564.304,A 0.000,B 0.000,C 90.000,E1 54.609} C_DIS
LIN {X -0.038,Y -285.034,Z 564.289,A 0.000,B 0.000,C 90.000,E1 51.949} C_DIS
LIN {X -0.035,Y -279.812,Z 564.277,A 0.000,B 0.000,C 90.000,E1 49.908} C_DIS
LIN {X 0.012,Y -274.134,Z 564.266,A 0.000,B 0.000,C 90.000,E1 47.838} C_DIS
LIN {X -0.016,Y -269.997,Z 564.258,A 0.000,B 0.000,C 90.000,E1 46.458} C_DIS
LIN {X 0.142,Y -264.394,Z 564.248,A 0.000,B 0.000,C 90.000,E1 44.676} C_DIS
LIN {X 0.118,Y -254.992,Z 564.233,A 0.000,B 0.000,C 90.000,E1 41.838} C_DIS
LIN {X -0.078,Y -244.928,Z 564.214,A 0.000,B 0.000,C 90.000,E1 38.624} C_DIS
LIN {X -0.071,Y -236.713,Z 564.198,A 0.000,B 0.000,C 90.000,E1 35.678} C_DIS
LIN {X -0.028,Y -229.171,Z 564.181,A 0.000,B 0.000,C 90.000,E1 32.673} C_DIS
LIN {X 0.035,Y -222.317,Z 564.165,A 0.000,B 0.000,C 90.000,E1 29.617} C_DIS
LIN {X 0.010,Y -216.258,Z 564.147,A 0.000,B 0.000,C 90.000,E1 26.539} C_DIS
LIN {X -0.033,Y -209.700,Z 564.126,A 0.000,B 0.000,C 90.000,E1 22.642} C_DIS
LIN {X 0.062,Y -205.652,Z 564.108,A 0.000,B 0.000,C 90.000,E1 19.450} C_DIS
LIN {X -0.034,Y -201.503,Z 564.086,A 0.000,B 0.000,C 90.000,E1 15.481} C_DIS
LIN {X 0.103,Y -197.882,Z 564.059,A 0.000,B 0.000,C 90.000,E1 10.602} C_DIS
LIN {X -0.045,Y -195.351,Z 564.018,A 0.000,B 0.000,C 90.000,E1 3.326} C_DIS
LIN {X 0.092,Y -197.142,Z 563.966,A 0.000,B 0.000,C 90.000,E1 353.799} C_DIS
LIN {X -0.084,Y -200.822,Z 563.934,A 0.000,B 0.000,C 90.000,E1 348.173} C_DIS
LIN {X 0.006,Y -205.342,Z 563.907,A 0.000,B 0.000,C 90.000,E1 343.323} C_DIS
LIN {X 0.018,Y -209.940,Z 563.885,A 0.000,B 0.000,C 90.000,E1 339.337} C_DIS
LIN {X -0.036,Y -215.272,Z 563.863,A 0.000,B 0.000,C 90.000,E1 335.409} C_DIS
LIN {X -0.039,Y -221.195,Z 563.842,A 0.000,B 0.000,C 90.000,E1 331.513} C_DIS
LIN {X -0.019,Y -227.731,Z 563.820,A 0.000,B 0.000,C 90.000,E1 327.661} C_DIS
LIN {X -0.007,Y -234.784,Z 563.799,A 0.000,B 0.000,C 90.000,E1 323.863} C_DIS
LIN {X 0.039,Y -242.366,Z 563.778,A 0.000,B 0.000,C 90.000,E1 320.114} C_DIS
LIN {X -0.073,Y -250.590,Z 563.758,A 0.000,B 0.000,C 90.000,E1 316.458} C_DIS
LIN {X -0.134,Y -260.167,Z 563.738,A 0.000,B 0.000,C 90.000,E1 312.852} C_DIS
LIN {X 0.010,Y -271.129,Z 563.718,A 0.000,B 0.000,C 90.000,E1 309.277} C_DIS
LIN {X 0.043,Y -283.631,Z 563.699,A 0.000,B 0.000,C 90.000,E1 305.804} C_DIS
LIN {X 0.055,Y -297.589,Z 563.680,A 0.000,B 0.000,C 90.000,E1 302.418} C_DIS
LIN {X -0.122,Y -312.735,Z 563.662,A 0.000,B 0.000,C 90.000,E1 299.155} C_DIS
LIN {X 0.007,Y -329.186,Z 563.644,A 0.000,B 0.000,C 90.000,E1 295.924} C_DIS
LIN {X -0.208,Y -341.849,Z 563.632,A 0.000,B 0.000,C 90.000,E1 293.770} C_DIS
LIN {X 0.023,Y -355.948,Z 563.620,A 0.000,B 0.000,C 90.000,E1 291.589} C_DIS
LIN {X 0.137,Y -378.099,Z 563.603,A 0.000,B 0.000,C 90.000,E1 288.598} C_DIS
END
